C03662=1159.444,359.025,-79.936,-176.298,9.017,148.740
C03663=1159.448,358.778,-79.901,-176.300,9.013,148.740
C03664=1159.452,358.530,-79.866,-176.303,9.010,148.739
C03665=1159.456,358.283,-79.832,-176.305,9.006,148.739
C03666=1159.460,358.035,-79.798,-176.307,9.002,148.739
C03667=1159.465,357.787,-79.763,-176.310,8.998,148.739
C03668=1159.467,357.540,-79.728,-176.313,8.995,148.738
C03669=1159.472,357.292,-79.694,-176.315,8.990,148.738
C03670=1159.476,357.044,-79.659,-176.317,8.987,148.738
C03671=1159.480,356.797,-79.625,-176.320,8.983,148.737
C03672=1159.484,356.549,-79.590,-176.322,8.979,148.737
C03673=1159.488,356.302,-79.556,-176.325,8.975,148.737
C03674=1159.492,356.054,-79.521,-176.327,8.972,148.736
C03675=1159.496,355.806,-79.487,-176.330,8.968,148.736
C03676=1159.499,355.559,-79.453,-176.332,8.964,148.736
C03677=1159.504,355.311,-79.418,-176.335,8.960,148.736
C03678=1159.508,355.064,-79.384,-176.337,8.957,148.735
C03679=1159.512,354.816,-79.350,-176.340,8.953,148.735
C03680=1159.516,354.569,-79.315,-176.342,8.949,148.735
C03681=1159.520,354.321,-79.281,-176.344,8.946,148.734
C03682=1159.524,354.073,-79.246,-176.347,8.942,148.734
C03683=1159.527,353.826,-79.212,-176.349,8.938,148.734
C03684=1159.532,353.578,-79.178,-176.352,8.934,148.733
C03685=1159.536,353.331,-79.144,-176.354,8.931,148.733
C03686=1159.540,353.083,-79.109,-176.357,8.926,148.733
C03687=1159.544,352.836,-79.075,-176.359,8.923,148.733
C03688=1159.548,352.588,-79.040,-176.362,8.919,148.732
C03689=1159.552,352.340,-79.007,-176.364,8.915,148.732
C03690=1159.556,352.093,-78.973,-176.366,8.912,148.732
C03691=1159.559,351.845,-78.938,-176.369,8.908,148.732
C03692=1159.564,351.597,-78.904,-176.372,8.905,148.731
C03693=1159.568,351.350,-78.870,-176.374,8.900,148.731
C03694=1159.571,351.102,-78.837,-176.376,8.897,148.731
C03695=1159.576,350.854,-78.802,-176.379,8.894,148.731
C03696=1159.579,350.607,-78.768,-176.382,8.890,148.730
C03697=1159.584,350.359,-78.733,-176.384,8.886,148.730
C03698=1159.588,350.111,-78.700,-176.387,8.882,148.730
C03699=1159.592,349.863,-78.665,-176.389,8.879,148.729
C03700=1159.596,349.616,-78.632,-176.391,8.875,148.729
C03701=1159.600,349.368,-78.598,-176.394,8.871,148.729
C03702=1159.604,349.121,-78.564,-176.396,8.868,148.729
C03703=1159.608,348.873,-78.530,-176.399,8.864,148.728
C03704=1159.612,348.625,-78.496,-176.401,8.861,148.728
C03705=1159.616,348.378,-78.462,-176.404,8.856,148.728
C03706=1159.620,348.130,-78.428,-176.406,8.853,148.728
C03707=1159.624,347.883,-78.395,-176.408,8.850,148.727
C03708=1159.628,347.635,-78.360,-176.411,8.846,148.727
C03709=1159.632,347.387,-78.327,-176.414,8.842,148.727
C03710=1159.636,347.140,-78.293,-176.416,8.838,148.727
C03711=1159.641,346.892,-78.259,-176.419,8.835,148.726
C03712=1159.644,346.644,-78.225,-176.421,8.832,148.726
C03713=1159.649,346.397,-78.192,-176.423,8.827,148.726
C03714=1159.652,346.149,-78.158,-176.426,8.824,148.726
C03715=1159.657,345.901,-78.124,-176.428,8.821,148.725
C03716=1159.660,345.654,-78.090,-176.431,8.817,148.725
C03717=1159.665,345.406,-78.057,-176.433,8.813,148.725
C03718=1159.668,345.158,-78.023,-176.436,8.809,148.725
C03719=1159.673,344.910,-77.989,-176.438,8.806,148.724
C03720=1159.677,344.662,-77.956,-176.441,8.803,148.724
C03721=1159.681,344.415,-77.922,-176.444,8.798,148.724
C03722=1159.685,344.168,-77.889,-176.446,8.795,148.724
C03723=1159.689,343.919,-77.854,-176.448,8.792,148.724
C03724=1159.693,343.672,-77.821,-176.451,8.788,148.723
C03725=1159.697,343.424,-77.788,-176.453,8.785,148.723
C03726=1159.701,343.177,-77.754,-176.456,8.780,148.723
C03727=1159.705,342.929,-77.721,-176.458,8.777,148.722
C03728=1159.709,342.681,-77.687,-176.461,8.774,148.722
C03729=1159.713,342.433,-77.653,-176.463,8.769,148.722
C03730=1159.717,342.186,-77.619,-176.466,8.766,148.722
C03731=1159.721,341.938,-77.586,-176.468,8.763,148.722
C03732=1159.726,341.690,-77.553,-176.471,8.759,148.721
C03733=1159.730,341.442,-77.520,-176.473,8.755,148.721
C03734=1159.734,341.195,-77.486,-176.475,8.752,148.721
C03735=1159.738,340.948,-77.453,-176.478,8.748,148.721
C03736=1159.741,340.699,-77.419,-176.481,8.745,148.720
C03737=1159.745,340.451,-77.386,-176.483,8.741,148.720
C03738=1159.749,340.204,-77.353,-176.486,8.737,148.720
C03739=1159.755,339.924,-77.315,-176.489,8.733,148.720
C03740=1159.759,339.644,-77.278,-176.492,8.729,148.719
C03741=1159.764,339.365,-77.240,-176.494,8.726,148.719
C03742=1159.769,339.085,-77.202,-176.497,8.722,148.719
C03743=1159.772,338.837,-77.169,-176.500,8.718,148.719
C03744=1159.776,338.589,-77.136,-176.502,8.714,148.718
C03745=1159.780,338.341,-77.103,-176.504,8.711,148.718
C03746=1159.785,338.093,-77.069,-176.507,8.707,148.718
C03747=1159.789,337.846,-77.036,-176.509,8.704,148.718
C03748=1159.793,337.598,-77.003,-176.512,8.700,148.718
C03749=1159.797,337.350,-76.970,-176.515,8.696,148.717
C03750=1159.801,337.102,-76.937,-176.517,8.693,148.717
C03751=1159.805,336.855,-76.904,-176.519,8.690,148.717
C03752=1159.809,336.607,-76.871,-176.523,8.686,148.717
C03753=1159.813,336.360,-76.838,-176.525,8.683,148.717
C03754=1159.817,336.112,-76.805,-176.527,8.679,148.717
C03755=1159.821,335.864,-76.772,-176.530,8.675,148.716
C03756=1159.825,335.616,-76.739,-176.532,8.672,148.716
C03757=1159.829,335.369,-76.705,-176.535,8.669,148.716
C03758=1159.834,335.120,-76.673,-176.537,8.665,148.716
C03759=1159.838,334.873,-76.640,-176.540,8.661,148.715
C03760=1159.841,334.625,-76.607,-176.542,8.658,148.715
C03761=1159.845,334.377,-76.574,-176.544,8.655,148.715
C03762=1159.850,334.130,-76.541,-176.547,8.651,148.715
C03763=1159.854,333.881,-76.508,-176.550,8.647,148.715
C03764=1159.858,333.634,-76.475,-176.552,8.644,148.714
C03765=1159.862,333.386,-76.442,-176.555,8.640,148.714
C03766=1159.866,333.138,-76.410,-176.558,8.637,148.714
C03767=1159.870,332.890,-76.377,-176.560,8.634,148.714
C03768=1159.874,332.642,-76.344,-176.562,8.630,148.714
C03769=1159.878,332.395,-76.311,-176.565,8.626,148.713
C03770=1159.883,332.147,-76.278,-176.567,8.623,148.713
C03771=1159.886,331.899,-76.246,-176.570,8.620,148.713
C03772=1159.890,331.651,-76.213,-176.573,8.616,148.713
C03773=1159.895,331.403,-76.179,-176.575,8.612,148.713
C03774=1159.898,331.155,-76.148,-176.578,8.609,148.713
C03775=1159.902,330.908,-76.114,-176.580,8.606,148.712
C03776=1159.907,330.659,-76.082,-176.583,8.602,148.712
C03777=1159.911,330.412,-76.049,-176.585,8.599,148.712
C03778=1159.915,330.165,-76.017,-176.587,8.595,148.712
C03779=1159.919,329.917,-75.984,-176.590,8.592,148.712
C03780=1159.924,329.669,-75.951,-176.593,8.588,148.711
C03781=1159.927,329.421,-75.919,-176.595,8.585,148.711
C03782=1159.931,329.173,-75.886,-176.598,8.582,148.711
C03783=1159.936,328.925,-75.854,-176.601,8.578,148.711
C03784=1159.939,328.677,-75.821,-176.603,8.574,148.711
C03785=1159.944,328.429,-75.789,-176.605,8.571,148.711
C03786=1159.948,328.182,-75.756,-176.607,8.568,148.710
C03787=1159.952,327.934,-75.724,-176.611,8.564,148.710
C03788=1159.956,327.686,-75.691,-176.613,8.561,148.710
C03789=1159.960,327.438,-75.659,-176.615,8.557,148.710
C03790=1159.964,327.190,-75.627,-176.618,8.554,148.710
C03791=1159.969,326.942,-75.593,-176.621,8.550,148.709
C03792=1159.973,326.695,-75.562,-176.623,8.547,148.709
C03793=1159.977,326.447,-75.529,-176.626,8.544,148.709
C03794=1159.981,326.199,-75.497,-176.628,8.541,148.709
C03795=1159.985,325.951,-75.465,-176.631,8.536,148.709
C03796=1159.989,325.703,-75.432,-176.633,8.533,148.709
C03797=1159.993,325.455,-75.400,-176.636,8.530,148.709
C03798=1159.997,325.207,-75.368,-176.638,8.527,148.708
C03799=1160.002,324.959,-75.336,-176.641,8.523,148.708
C03800=1160.005,324.712,-75.303,-176.643,8.520,148.708
C03801=1160.010,324.463,-75.271,-176.646,8.517,148.708
C03802=1160.013,324.215,-75.239,-176.648,8.513,148.708
C03803=1160.018,323.968,-75.206,-176.651,8.510,148.708
C03804=1160.022,323.720,-75.174,-176.654,8.506,148.707
C03805=1160.026,323.472,-75.142,-176.656,8.503,148.707
C03806=1160.030,323.224,-75.110,-176.659,8.500,148.707
C03807=1160.035,322.976,-75.078,-176.661,8.496,148.707
C03808=1160.039,322.728,-75.046,-176.664,8.492,148.707
C03809=1160.042,322.481,-75.013,-176.666,8.489,148.707
C03810=1160.047,322.232,-74.981,-176.669,8.486,148.707
C03811=1160.051,321.985,-74.949,-176.671,8.483,148.706
C03812=1160.055,321.737,-74.917,-176.674,8.479,148.706
C03813=1160.059,321.489,-74.885,-176.677,8.476,148.706
C03814=1160.063,321.241,-74.853,-176.679,8.472,148.706
C03815=1160.068,320.993,-74.821,-176.681,8.469,148.706
C03816=1160.071,320.745,-74.789,-176.684,8.466,148.706
C03817=1160.075,320.497,-74.758,-176.687,8.462,148.706
C03818=1160.080,320.249,-74.725,-176.689,8.459,148.705
C03819=1160.084,320.001,-74.694,-176.692,8.455,148.705
C03820=1160.088,319.753,-74.662,-176.694,8.452,148.705
C03821=1160.093,319.506,-74.630,-176.697,8.449,148.705
C03822=1160.096,319.257,-74.598,-176.700,8.445,148.705
C03823=1160.100,319.009,-74.566,-176.702,8.442,148.705
C03824=1160.105,318.762,-74.534,-176.705,8.439,148.705
C03825=1160.109,318.514,-74.502,-176.707,8.436,148.704
C03826=1160.113,318.266,-74.470,-176.709,8.432,148.704
C03827=1160.117,318.018,-74.439,-176.713,8.428,148.704
C03828=1160.121,317.770,-74.406,-176.715,8.425,148.704
C03829=1160.125,317.522,-74.374,-176.717,8.422,148.704
C03830=1160.130,317.274,-74.344,-176.720,8.419,148.704
C03831=1160.133,317.026,-74.312,-176.722,8.416,148.704
C03832=1160.137,316.778,-74.280,-176.725,8.412,148.703
C03833=1160.142,316.530,-74.248,-176.728,8.409,148.703
C03834=1160.146,316.282,-74.216,-176.730,8.405,148.703
C03835=1160.150,316.035,-74.185,-176.732,8.402,148.703
C03836=1160.154,315.786,-74.153,-176.735,8.399,148.703
C03837=1160.158,315.538,-74.122,-176.738,8.395,148.703
C03838=1160.163,315.291,-74.090,-176.740,8.392,148.703
C03839=1160.167,315.043,-74.058,-176.743,8.389,148.703
C03840=1160.171,314.795,-74.027,-176.745,8.385,148.702
C03841=1160.175,314.547,-73.995,-176.748,8.382,148.702
C03842=1160.179,314.299,-73.964,-176.750,8.379,148.702
C03843=1160.184,314.021,-73.929,-176.753,8.375,148.702
C03844=1160.189,313.744,-73.894,-176.757,8.371,148.702
C03845=1160.193,313.467,-73.858,-176.759,8.368,148.702
C03846=1160.198,313.190,-73.823,-176.762,8.364,148.702
C03847=1160.202,312.941,-73.792,-176.765,8.361,148.702
C03848=1160.206,312.694,-73.760,-176.767,8.358,148.701
C03849=1160.210,312.446,-73.728,-176.770,8.354,148.701
C03850=1160.215,312.198,-73.697,-176.773,8.351,148.701
C03851=1160.218,311.950,-73.666,-176.775,8.347,148.701
C03852=1160.223,311.702,-73.635,-176.778,8.344,148.701
C03853=1160.227,311.454,-73.603,-176.780,8.341,148.701
C03854=1160.231,311.206,-73.572,-176.783,8.338,148.701
C03855=1160.235,310.958,-73.540,-176.786,8.334,148.701
C03856=1160.240,310.710,-73.510,-176.788,8.331,148.700
C03857=1160.243,310.462,-73.478,-176.791,8.328,148.700
C03858=1160.248,310.214,-73.447,-176.793,8.324,148.700
C03859=1160.252,309.966,-73.415,-176.796,8.321,148.700
C03860=1160.256,309.718,-73.384,-176.798,8.318,148.700
C03861=1160.260,309.469,-73.353,-176.800,8.315,148.700
C03862=1160.264,309.222,-73.322,-176.804,8.311,148.700
C03863=1160.268,308.973,-73.291,-176.806,8.308,148.700
C03864=1160.273,308.726,-73.259,-176.809,8.305,148.700
C03865=1160.277,308.477,-73.228,-176.811,8.302,148.700
C03866=1160.281,308.229,-73.197,-176.814,8.299,148.700
C03867=1160.286,307.982,-73.166,-176.816,8.295,148.699
C03868=1160.290,307.733,-73.135,-176.818,8.292,148.699
C03869=1160.294,307.485,-73.104,-176.822,8.288,148.699
C03870=1160.298,307.237,-73.072,-176.824,8.285,148.699
C03871=1160.302,306.990,-73.042,-176.827,8.282,148.699
C03872=1160.307,306.742,-73.011,-176.829,8.279,148.699
C03873=1160.311,306.493,-72.980,-176.832,8.276,148.699
C03874=1160.315,306.246,-72.949,-176.834,8.272,148.699
C03875=1160.319,305.997,-72.917,-176.837,8.269,148.699
C03876=1160.323,305.749,-72.887,-176.839,8.266,148.699
C03877=1160.328,305.501,-72.856,-176.842,8.262,148.698
C03878=1160.331,305.253,-72.825,-176.845,8.259,148.698
C03879=1160.336,305.005,-72.794,-176.847,8.256,148.698
C03880=1160.340,304.757,-72.763,-176.850,8.253,148.698
C03881=1160.344,304.509,-72.732,-176.853,8.250,148.698
C03882=1160.349,304.261,-72.701,-176.855,8.247,148.698
C03883=1160.353,304.013,-72.671,-176.858,8.244,148.698
C03884=1160.357,303.765,-72.640,-176.860,8.240,148.698
C03885=1160.361,303.517,-72.609,-176.863,8.237,148.698
C03886=1160.366,303.269,-72.578,-176.866,8.233,148.698
C03887=1160.369,303.020,-72.548,-176.868,8.230,148.698
C03888=1160.374,302.772,-72.517,-176.871,8.227,148.697
C03889=1160.378,302.525,-72.486,-176.873,8.224,148.698
C03890=1160.382,302.276,-72.454,-176.876,8.221,148.697
C03891=1160.386,302.029,-72.424,-176.878,8.218,148.697
C03892=1160.391,301.781,-72.394,-176.881,8.215,148.697
C03893=1160.395,301.533,-72.363,-176.883,8.212,148.697
C03894=1160.399,301.284,-72.333,-176.886,8.208,148.697
C03895=1160.404,301.036,-72.302,-176.889,8.205,148.697
C03896=1160.408,300.788,-72.271,-176.891,8.201,148.697
C03897=1160.411,300.540,-72.241,-176.894,8.198,148.697
C03898=1160.416,300.292,-72.210,-176.896,8.195,148.697
C03899=1160.421,300.044,-72.179,-176.899,8.192,148.697
C03900=1160.425,299.796,-72.149,-176.901,8.189,148.697
C03901=1160.429,299.547,-72.118,-176.904,8.186,148.697
C03902=1160.433,299.299,-72.087,-176.907,8.183,148.696
C03903=1160.437,299.052,-72.057,-176.909,8.180,148.696
C03904=1160.442,298.803,-72.027,-176.912,8.177,148.696
C03905=1160.445,298.555,-71.997,-176.914,8.173,148.696
C03906=1160.450,298.307,-71.966,-176.918,8.170,148.696
C03907=1160.454,298.059,-71.935,-176.920,8.166,148.696
C03908=1160.458,297.811,-71.905,-176.923,8.163,148.696
C03909=1160.463,297.563,-71.875,-176.925,8.160,148.696
C03910=1160.467,297.314,-71.844,-176.928,8.157,148.696
C03911=1160.471,297.066,-71.813,-176.931,8.154,148.696
C03912=1160.475,296.818,-71.784,-176.933,8.151,148.696
C03913=1160.480,296.570,-71.753,-176.936,8.148,148.696
C03914=1160.484,296.322,-71.723,-176.938,8.145,148.696
C03915=1160.488,296.074,-71.692,-176.941,8.142,148.696
C03916=1160.492,295.826,-71.663,-176.943,8.138,148.695
C03917=1160.497,295.578,-71.632,-176.946,8.135,148.696
C03918=1160.500,295.330,-71.602,-176.948,8.132,148.696
C03919=1160.505,295.081,-71.572,-176.951,8.128,148.695
C03920=1160.509,294.834,-71.541,-176.954,8.125,148.695
C03921=1160.513,294.585,-71.512,-176.956,8.122,148.695
C03922=1160.517,294.337,-71.481,-176.959,8.119,148.695
C03923=1160.521,294.089,-71.451,-176.962,8.116,148.695
C03924=1160.526,293.841,-71.421,-176.964,8.113,148.695
C03925=1160.530,293.593,-71.390,-176.967,8.110,148.695
C03926=1160.534,293.345,-71.361,-176.970,8.107,148.695
C03927=1160.539,293.097,-71.330,-176.972,8.104,148.695
C03928=1160.543,292.848,-71.301,-176.975,8.101,148.695
C03929=1160.547,292.600,-71.270,-176.977,8.097,148.695
C03930=1160.551,292.351,-71.240,-176.980,8.094,148.695
C03931=1160.555,292.104,-71.210,-176.983,8.091,148.695
C03932=1160.560,291.855,-71.180,-176.985,8.088,148.695
C03933=1160.564,291.607,-71.150,-176.988,8.085,148.695
C03934=1160.568,291.359,-71.120,-176.990,8.082,148.695
C03935=1160.573,291.111,-71.090,-176.993,8.079,148.695
C03936=1160.577,290.863,-71.060,-176.995,8.076,148.695
C03937=1160.581,290.615,-71.031,-176.998,8.073,148.695
C03938=1160.585,290.367,-71.001,-177.001,8.069,148.694
C03939=1160.590,290.119,-70.970,-177.004,8.066,148.695
C03940=1160.594,289.870,-70.941,-177.007,8.063,148.695
C03941=1160.598,289.622,-70.912,-177.009,8.060,148.694
C03942=1160.603,289.374,-70.881,-177.012,8.057,148.694
C03943=1160.607,289.126,-70.851,-177.014,8.054,148.694
C03944=1160.611,288.878,-70.822,-177.017,8.051,148.694
C03945=1160.615,288.630,-70.792,-177.019,8.048,148.694
C03946=1160.619,288.382,-70.762,-177.022,8.045,148.694
C03947=1160.624,288.106,-70.729,-177.025,8.041,148.694
C03948=1160.628,287.831,-70.696,-177.028,8.038,148.694
C03949=1160.633,287.555,-70.663,-177.031,8.035,148.694
C03950=1160.638,287.281,-70.630,-177.034,8.031,148.694
C03951=1160.642,287.032,-70.601,-177.036,8.028,148.694
C03952=1160.647,286.784,-70.571,-177.039,8.025,148.694
C03953=1160.651,286.536,-70.541,-177.042,8.022,148.694
C03954=1160.656,286.289,-70.511,-177.044,8.018,148.694
C03955=1160.660,286.040,-70.482,-177.047,8.015,148.694
C03956=1160.664,285.792,-70.452,-177.050,8.012,148.694
C03957=1160.668,285.544,-70.423,-177.052,8.009,148.694
C03958=1160.672,285.296,-70.393,-177.055,8.006,148.694
C03959=1160.677,285.047,-70.363,-177.057,8.003,148.694
C03960=1160.681,284.799,-70.334,-177.060,8.000,148.694
C03961=1160.686,284.550,-70.304,-177.062,7.997,148.694
C03962=1160.690,284.302,-70.275,-177.065,7.994,148.694
C03963=1160.694,284.054,-70.246,-177.068,7.991,148.694
C03964=1160.698,283.806,-70.216,-177.071,7.988,148.694
C03965=1160.702,283.557,-70.187,-177.073,7.985,148.694
C03966=1160.707,283.309,-70.157,-177.076,7.982,148.694
C03967=1160.711,283.061,-70.128,-177.079,7.979,148.694
C03968=1160.716,282.813,-70.099,-177.081,7.976,148.694
C03969=1160.720,282.565,-70.069,-177.084,7.973,148.694
C03970=1160.724,282.317,-70.040,-177.086,7.970,148.694
C03971=1160.728,282.068,-70.010,-177.089,7.967,148.694
C03972=1160.732,281.820,-69.981,-177.092,7.964,148.694
C03973=1160.736,281.572,-69.951,-177.094,7.961,148.694
C03974=1160.741,281.324,-69.922,-177.097,7.958,148.694
C03975=1160.746,281.076,-69.894,-177.100,7.955,148.694
C03976=1160.750,280.827,-69.864,-177.102,7.952,148.694
C03977=1160.754,280.579,-69.835,-177.105,7.948,148.694
C03978=1160.758,280.331,-69.805,-177.108,7.945,148.694
C03979=1160.762,280.082,-69.776,-177.110,7.942,148.694
C03980=1160.767,279.834,-69.746,-177.113,7.940,148.694
C03981=1160.771,279.585,-69.718,-177.115,7.936,148.694
C03982=1160.776,279.338,-69.688,-177.118,7.933,148.694
C03983=1160.780,279.089,-69.659,-177.121,7.930,148.694
C03984=1160.784,278.841,-69.630,-177.124,7.927,148.694
C03985=1160.788,278.593,-69.601,-177.126,7.924,148.694
C03986=1160.792,278.344,-69.572,-177.128,7.922,148.694
C03987=1160.797,278.097,-69.543,-177.131,7.919,148.694
C03988=1160.801,277.848,-69.514,-177.134,7.916,148.694
C03989=1160.806,277.600,-69.485,-177.136,7.913,148.694
C03990=1160.810,277.351,-69.455,-177.139,7.910,148.694
C03991=1160.814,277.103,-69.427,-177.141,7.907,148.694
C03992=1160.818,276.855,-69.398,-177.144,7.904,148.694
C03993=1160.823,276.607,-69.369,-177.147,7.901,148.694
C03994=1160.827,276.358,-69.340,-177.150,7.898,148.694
C03995=1160.831,276.110,-69.310,-177.152,7.895,148.694
C03996=1160.836,275.862,-69.283,-177.155,7.892,148.694
C03997=1160.840,275.614,-69.253,-177.158,7.889,148.694
C03998=1160.844,275.365,-69.224,-177.160,7.886,148.694
C03999=1160.848,275.116,-69.195,-177.163,7.883,148.694
C04000=1160.852,274.869,-69.166,-177.166,7.880,148.694
C04001=1160.857,274.620,-69.138,-177.169,7.877,148.694
C04002=1160.861,274.372,-69.108,-177.171,7.874,148.694
C04003=1160.866,274.124,-69.080,-177.174,7.871,148.694
C04004=1160.870,273.876,-69.051,-177.176,7.868,148.694
C04005=1160.874,273.627,-69.022,-177.179,7.865,148.694
C04006=1160.878,273.379,-68.993,-177.182,7.862,148.694
C04007=1160.883,273.131,-68.965,-177.185,7.859,148.694
C04008=1160.887,272.882,-68.936,-177.187,7.857,148.694
C04009=1160.891,272.634,-68.907,-177.189,7.853,148.694
C04010=1160.896,272.386,-68.879,-177.192,7.851,148.694
C04011=1160.900,272.138,-68.850,-177.195,7.848,148.694
C04012=1160.904,271.889,-68.821,-177.197,7.845,148.694
C04013=1160.909,271.641,-68.793,-177.200,7.842,148.694
C04014=1160.913,271.393,-68.764,-177.203,7.839,148.694
C04015=1160.917,271.144,-68.735,-177.206,7.836,148.694
C04016=1160.922,270.896,-68.707,-177.208,7.833,148.694
C04017=1160.926,270.648,-68.678,-177.211,7.830,148.694
C04018=1160.931,270.399,-68.649,-177.214,7.827,148.694
C04019=1160.935,270.151,-68.621,-177.216,7.824,148.694
C04020=1160.939,269.902,-68.592,-177.219,7.821,148.694
C04021=1160.943,269.655,-68.564,-177.222,7.818,148.694
C04022=1160.948,269.406,-68.535,-177.224,7.816,148.694
C04023=1160.952,269.157,-68.507,-177.227,7.813,148.694
C04024=1160.957,268.909,-68.479,-177.230,7.810,148.695
C04025=1160.960,268.660,-68.451,-177.232,7.807,148.695
C04026=1160.965,268.413,-68.421,-177.235,7.804,148.695
C04027=1160.970,268.164,-68.393,-177.237,7.800,148.694
C04028=1160.974,267.916,-68.365,-177.240,7.798,148.695
C04029=1160.978,267.667,-68.336,-177.243,7.795,148.695
C04030=1160.982,267.419,-68.308,-177.246,7.792,148.695
C04031=1160.987,267.170,-68.280,-177.248,7.789,148.695
C04032=1160.991,266.922,-68.252,-177.251,7.786,148.695
C04033=1160.996,266.674,-68.223,-177.253,7.784,148.695
C04034=1161.000,266.426,-68.194,-177.256,7.781,148.695
C04035=1161.004,266.178,-68.167,-177.259,7.778,148.695
C04036=1161.008,265.929,-68.138,-177.262,7.775,148.695
C04037=1161.013,265.681,-68.110,-177.264,7.772,148.695
C04038=1161.017,265.432,-68.081,-177.267,7.769,148.695
C04039=1161.022,265.184,-68.054,-177.270,7.766,148.695
C04040=1161.026,264.935,-68.025,-177.273,7.763,148.695
C04041=1161.030,264.688,-67.997,-177.275,7.760,148.695
C04042=1161.034,264.439,-67.969,-177.278,7.757,148.695
C04043=1161.039,264.191,-67.941,-177.280,7.755,148.695
C04044=1161.043,263.942,-67.912,-177.283,7.752,148.695
C04045=1161.048,263.693,-67.885,-177.285,7.749,148.695
C04046=1161.052,263.445,-67.857,-177.288,7.746,148.695
C04047=1161.057,263.197,-67.829,-177.291,7.743,148.695
C04048=1161.061,262.948,-67.800,-177.294,7.740,148.695
C04049=1161.065,262.700,-67.772,-177.296,7.737,148.696
C04050=1161.069,262.452,-67.744,-177.299,7.734,148.696
C04051=1161.074,262.178,-67.713,-177.302,7.731,148.696
C04052=1161.080,261.905,-67.683,-177.305,7.728,148.696
C04053=1161.084,261.632,-67.652,-177.308,7.725,148.696
C04054=1161.089,261.359,-67.621,-177.311,7.721,148.696
C04055=1161.093,261.110,-67.593,-177.313,7.719,148.696
C04056=1161.097,260.862,-67.565,-177.316,7.716,148.696
C04057=1161.102,260.613,-67.537,-177.319,7.713,148.696
C04058=1161.106,260.365,-67.509,-177.321,7.710,148.696
C04059=1161.111,260.117,-67.482,-177.324,7.707,148.696
C04060=1161.114,259.868,-67.454,-177.327,7.704,148.696
C04061=1161.119,259.621,-67.426,-177.330,7.701,148.696
C04062=1161.124,259.371,-67.398,-177.332,7.699,148.696
C04063=1161.128,259.123,-67.370,-177.335,7.696,148.696
C04064=1161.132,258.875,-67.342,-177.337,7.693,148.696
C04065=1161.136,258.626,-67.315,-177.341,7.691,148.697
C04066=1161.141,258.378,-67.287,-177.343,7.688,148.697
C04067=1161.146,258.130,-67.259,-177.346,7.685,148.697
C04068=1161.150,257.881,-67.231,-177.349,7.682,148.697
C04069=1161.154,257.633,-67.203,-177.351,7.680,148.697
C04070=1161.158,257.384,-67.176,-177.354,7.677,148.697
C04071=1161.163,257.136,-67.148,-177.357,7.674,148.697
C04072=1161.167,256.888,-67.120,-177.359,7.671,148.697
C04073=1161.172,256.638,-67.092,-177.362,7.668,148.697
C04074=1161.176,256.391,-67.065,-177.365,7.665,148.697
C04075=1161.181,256.142,-67.038,-177.367,7.663,148.697
C04076=1161.185,255.894,-67.009,-177.370,7.660,148.697
C04077=1161.189,255.645,-66.982,-177.373,7.657,148.697
C04078=1161.194,255.397,-66.955,-177.375,7.654,148.698
C04079=1161.198,255.149,-66.928,-177.378,7.651,148.698
C04080=1161.202,254.900,-66.899,-177.381,7.648,148.698
C04081=1161.207,254.652,-66.872,-177.383,7.646,148.698
C04082=1161.211,254.403,-66.845,-177.386,7.643,148.698
C04083=1161.215,254.154,-66.817,-177.389,7.640,148.698
C04084=1161.220,253.906,-66.790,-177.391,7.637,148.698
C04085=1161.224,253.658,-66.762,-177.394,7.634,148.698
C04086=1161.229,253.410,-66.735,-177.397,7.632,148.698
C04087=1161.233,253.160,-66.708,-177.400,7.629,148.698
C04088=1161.237,252.913,-66.680,-177.402,7.627,148.698
C04089=1161.242,252.664,-66.653,-177.405,7.624,148.699
C04090=1161.246,252.415,-66.626,-177.408,7.621,148.699
C04091=1161.250,252.167,-66.598,-177.411,7.618,148.699
C04092=1161.255,251.918,-66.571,-177.413,7.616,148.699
C04093=1161.259,251.670,-66.544,-177.416,7.613,148.699
C04094=1161.264,251.422,-66.516,-177.418,7.610,148.699
C04095=1161.268,251.173,-66.488,-177.421,7.607,148.699
C04096=1161.273,250.924,-66.461,-177.424,7.604,148.699
C04097=1161.277,250.676,-66.434,-177.427,7.602,148.699
C04098=1161.282,250.428,-66.407,-177.429,7.599,148.699
C04099=1161.286,250.179,-66.379,-177.432,7.596,148.699
C04100=1161.290,249.930,-66.352,-177.435,7.593,148.700
C04101=1161.294,249.682,-66.326,-177.438,7.590,148.700
C04102=1161.299,249.434,-66.299,-177.440,7.588,148.700
C04103=1161.303,249.186,-66.271,-177.443,7.585,148.700
C04104=1161.308,248.937,-66.244,-177.445,7.582,148.700
C04105=1161.312,248.688,-66.216,-177.449,7.580,148.700
C04106=1161.317,248.440,-66.189,-177.451,7.577,148.700
C04107=1161.321,248.191,-66.162,-177.454,7.574,148.700
C04108=1161.325,247.943,-66.136,-177.456,7.572,148.700
C04109=1161.330,247.694,-66.109,-177.459,7.569,148.700
C04110=1161.334,247.446,-66.082,-177.462,7.566,148.700
C04111=1161.338,247.197,-66.054,-177.464,7.564,148.701
C04112=1161.343,246.948,-66.027,-177.467,7.561,148.701
C04113=1161.347,246.700,-66.001,-177.470,7.558,148.701
C04114=1161.352,246.452,-65.974,-177.473,7.555,148.701
C04115=1161.356,246.203,-65.946,-177.476,7.552,148.701
C04116=1161.361,245.955,-65.919,-177.478,7.550,148.701
C04117=1161.366,245.706,-65.892,-177.481,7.547,148.701
C04118=1161.370,245.458,-65.866,-177.483,7.544,148.701
C04119=1161.374,245.209,-65.839,-177.487,7.541,148.702
C04120=1161.378,244.960,-65.811,-177.489,7.539,148.702
C04121=1161.382,244.712,-65.785,-177.491,7.536,148.702
C04122=1161.387,244.464,-65.758,-177.494,7.533,148.702
C04123=1161.392,244.215,-65.731,-177.497,7.530,148.702
C04124=1161.395,243.967,-65.704,-177.499,7.528,148.702
C04125=1161.400,243.718,-65.677,-177.502,7.526,148.702
C04126=1161.405,243.470,-65.650,-177.505,7.523,148.702
C04127=1161.409,243.221,-65.624,-177.508,7.520,148.702
C04128=1161.414,242.973,-65.597,-177.510,7.518,148.703
C04129=1161.418,242.724,-65.570,-177.513,7.515,148.703
C04130=1161.422,242.476,-65.544,-177.516,7.512,148.703
C04131=1161.427,242.227,-65.517,-177.519,7.509,148.703
C04132=1161.432,241.978,-65.490,-177.521,7.507,148.703
C04133=1161.436,241.730,-65.464,-177.524,7.504,148.703
C04134=1161.440,241.482,-65.437,-177.527,7.501,148.703
C04135=1161.444,241.233,-65.410,-177.530,7.499,148.704
C04136=1161.449,240.984,-65.384,-177.532,7.496,148.704
C04137=1161.454,240.736,-65.357,-177.535,7.494,148.704
C04138=1161.458,240.488,-65.331,-177.538,7.491,148.704
C04139=1161.463,240.239,-65.304,-177.540,7.488,148.704
C04140=1161.467,239.990,-65.278,-177.543,7.486,148.704
C04141=1161.471,239.742,-65.251,-177.546,7.483,148.704
C04142=1161.475,239.494,-65.224,-177.549,7.480,148.704
C04143=1161.480,239.245,-65.198,-177.551,7.478,148.704
C04144=1161.484,238.996,-65.171,-177.554,7.475,148.705
C04145=1161.489,238.747,-65.145,-177.557,7.472,148.705
C04146=1161.494,238.499,-65.118,-177.560,7.469,148.705
C04147=1161.498,238.251,-65.092,-177.562,7.467,148.705
C04148=1161.502,238.002,-65.066,-177.565,7.465,148.705
C04149=1161.507,237.753,-65.039,-177.568,7.462,148.705
C04150=1161.511,237.504,-65.013,-177.570,7.460,148.705
C04151=1161.516,237.256,-64.986,-177.573,7.457,148.706
C04152=1161.520,237.007,-64.960,-177.576,7.454,148.706
C04153=1161.524,236.759,-64.933,-177.578,7.452,148.706
C04154=1161.529,236.510,-64.907,-177.581,7.449,148.706
C04155=1161.534,236.238,-64.878,-177.584,7.446,148.706
C04156=1161.538,235.967,-64.849,-177.587,7.443,148.706
C04157=1161.544,235.695,-64.821,-177.590,7.440,148.706
C04158=1161.548,235.423,-64.792,-177.593,7.438,148.707
C04159=1161.553,235.174,-64.766,-177.596,7.435,148.707
C04160=1161.557,234.927,-64.739,-177.598,7.432,148.707
C04161=1161.562,234.678,-64.714,-177.601,7.430,148.707
C04162=1161.567,234.429,-64.687,-177.604,7.427,148.707
C04163=1161.571,234.181,-64.661,-177.607,7.424,148.707
C04164=1161.575,233.932,-64.635,-177.609,7.422,148.707
C04165=1161.580,233.683,-64.609,-177.612,7.420,148.708
C04166=1161.584,233.435,-64.582,-177.615,7.417,148.708
C04167=1161.588,233.187,-64.557,-177.618,7.414,148.708
C04168=1161.593,232.937,-64.531,-177.620,7.412,148.708
C04169=1161.597,232.689,-64.504,-177.623,7.409,148.708
C04170=1161.602,232.440,-64.478,-177.626,7.406,148.708
C04171=1161.607,232.191,-64.452,-177.628,7.404,148.709
C04172=1161.610,231.943,-64.426,-177.631,7.401,148.709
C04173=1161.615,231.695,-64.400,-177.634,7.398,148.709
C04174=1161.620,231.446,-64.374,-177.636,7.396,148.709
C04175=1161.624,231.197,-64.348,-177.639,7.394,148.709
C04176=1161.628,230.949,-64.322,-177.642,7.391,148.709
C04177=1161.633,230.700,-64.296,-177.644,7.389,148.710
C04178=1161.637,230.452,-64.270,-177.647,7.386,148.710
C04179=1161.642,230.203,-64.244,-177.650,7.384,148.710
C04180=1161.647,229.954,-64.218,-177.653,7.381,148.710
C04181=1161.651,229.705,-64.193,-177.655,7.378,148.710
C04182=1161.655,229.458,-64.167,-177.658,7.376,148.710
C04183=1161.660,229.209,-64.141,-177.661,7.373,148.711
C04184=1161.665,228.960,-64.114,-177.664,7.370,148.711
C04185=1161.669,228.711,-64.089,-177.666,7.368,148.711
C04186=1161.673,228.462,-64.063,-177.669,7.366,148.711
C04187=1161.678,228.214,-64.038,-177.672,7.363,148.711
C04188=1161.682,227.965,-64.012,-177.675,7.361,148.711
C04189=1161.686,227.717,-63.986,-177.677,7.358,148.711
C04190=1161.691,227.468,-63.961,-177.681,7.355,148.712
C04191=1161.696,227.219,-63.934,-177.683,7.353,148.712
C04192=1161.700,226.971,-63.909,-177.686,7.350,148.712
C04193=1161.705,226.722,-63.883,-177.688,7.348,148.712
C04194=1161.709,226.474,-63.857,-177.691,7.345,148.712
C04195=1161.714,226.225,-63.832,-177.694,7.343,148.712
C04196=1161.718,225.976,-63.806,-177.696,7.341,148.713
C04197=1161.723,225.728,-63.781,-177.699,7.338,148.713
C04198=1161.727,225.479,-63.755,-177.702,7.335,148.713
C04199=1161.731,225.230,-63.729,-177.705,7.333,148.713
C04200=1161.736,224.982,-63.704,-177.707,7.330,148.713
C04201=1161.740,224.733,-63.678,-177.710,7.328,148.714
C04202=1161.744,224.485,-63.652,-177.713,7.325,148.714
C04203=1161.749,224.237,-63.627,-177.716,7.322,148.714
C04204=1161.754,223.987,-63.602,-177.718,7.321,148.714
C04205=1161.758,223.738,-63.576,-177.721,7.318,148.714
C04206=1161.763,223.490,-63.551,-177.723,7.316,148.714
C04207=1161.767,223.241,-63.525,-177.726,7.313,148.715
C04208=1161.771,222.993,-63.499,-177.729,7.310,148.715
C04209=1161.776,222.744,-63.474,-177.732,7.308,148.715
C04210=1161.781,222.495,-63.449,-177.735,7.305,148.715
C04211=1161.785,222.247,-63.423,-177.737,7.303,148.715
C04212=1161.790,221.998,-63.398,-177.740,7.301,148.716
C04213=1161.794,221.749,-63.372,-177.743,7.298,148.716
C04214=1161.799,221.501,-63.347,-177.746,7.296,148.716
C04215=1161.803,221.252,-63.321,-177.748,7.293,148.716
C04216=1161.808,221.004,-63.296,-177.751,7.291,148.716
C04217=1161.813,220.754,-63.271,-177.754,7.288,148.717
C04218=1161.817,220.505,-63.245,-177.756,7.286,148.717
C04219=1161.822,220.257,-63.220,-177.759,7.284,148.717
C04220=1161.826,220.008,-63.195,-177.762,7.281,148.717
C04221=1161.830,219.760,-63.170,-177.764,7.279,148.717
C04222=1161.834,219.511,-63.144,-177.767,7.276,148.718
C04223=1161.839,219.262,-63.119,-177.770,7.274,148.718
C04224=1161.844,219.014,-63.094,-177.773,7.271,148.718
C04225=1161.848,218.765,-63.068,-177.775,7.269,148.718
C04226=1161.853,218.516,-63.043,-177.778,7.266,148.718
C04227=1161.857,218.268,-63.018,-177.781,7.264,148.718
C04228=1161.862,218.019,-62.994,-177.783,7.261,148.719
C04229=1161.866,217.770,-62.968,-177.787,7.259,148.719
C04230=1161.871,217.522,-62.943,-177.789,7.257,148.719
C04231=1161.875,217.273,-62.917,-177.792,7.254,148.719
C04232=1161.880,217.024,-62.893,-177.794,7.252,148.719
C04233=1161.884,216.776,-62.868,-177.797,7.249,148.720
C04234=1161.889,216.527,-62.843,-177.800,7.247,148.720
C04235=1161.893,216.278,-62.817,-177.803,7.245,148.720
C04236=1161.898,216.030,-62.793,-177.806,7.242,148.720
C04237=1161.902,215.781,-62.767,-177.808,7.240,148.720
C04238=1161.907,215.532,-62.743,-177.811,7.237,148.721
C04239=1161.911,215.283,-62.717,-177.813,7.235,148.721
C04240=1161.916,215.035,-62.693,-177.817,7.232,148.721
C04241=1161.920,214.785,-62.668,-177.819,7.230,148.721
C04242=1161.925,214.537,-62.642,-177.822,7.228,148.722
C04243=1161.929,214.288,-62.618,-177.824,7.226,148.722
C04244=1161.934,214.040,-62.593,-177.827,7.223,148.722
C04245=1161.938,213.791,-62.568,-177.830,7.221,148.722
C04246=1161.943,213.542,-62.543,-177.833,7.218,148.722
C04247=1161.947,213.294,-62.518,-177.835,7.216,148.723
C04248=1161.952,213.045,-62.493,-177.838,7.213,148.723
C04249=1161.956,212.796,-62.469,-177.841,7.211,148.723
C04250=1161.961,212.547,-62.444,-177.844,7.209,148.723
C04251=1161.966,212.299,-62.419,-177.846,7.207,148.723
C04252=1161.970,212.050,-62.394,-177.849,7.204,148.724
C04253=1161.975,211.801,-62.369,-177.851,7.202,148.724
C04254=1161.979,211.553,-62.345,-177.855,7.199,148.724
C04255=1161.983,211.304,-62.320,-177.857,7.197,148.724
C04256=1161.988,211.055,-62.295,-177.860,7.195,148.725
C04257=1161.993,210.807,-62.271,-177.862,7.193,148.725
C04258=1161.997,210.557,-62.246,-177.866,7.190,148.725
C04259=1162.002,210.287,-62.219,-177.868,7.187,148.725
C04260=1162.007,210.016,-62.192,-177.872,7.184,148.725
C04261=1162.012,209.746,-62.165,-177.874,7.182,148.726
C04262=1162.017,209.476,-62.139,-177.877,7.180,148.726
C04263=1162.021,209.227,-62.114,-177.880,7.177,148.726
C04264=1162.026,208.978,-62.090,-177.883,7.175,148.726
C04265=1162.031,208.730,-62.065,-177.886,7.172,148.727
C04266=1162.035,208.480,-62.040,-177.888,7.170,148.727
C04267=1162.040,208.232,-62.016,-177.891,7.168,148.727
C04268=1162.045,207.983,-61.992,-177.893,7.166,148.727
C04269=1162.048,207.734,-61.967,-177.897,7.163,148.728
C04270=1162.053,207.486,-61.942,-177.899,7.161,148.728
C04271=1162.058,207.237,-61.918,-177.902,7.159,148.728
C04272=1162.062,206.988,-61.893,-177.904,7.156,148.728
C04273=1162.067,206.739,-61.869,-177.907,7.154,148.728
C04274=1162.072,206.491,-61.844,-177.910,7.151,148.729
C04275=1162.076,206.242,-61.820,-177.912,7.150,148.729
C04276=1162.081,205.992,-61.796,-177.915,7.147,148.729
C04277=1162.085,205.744,-61.772,-177.918,7.145,148.729
C04278=1162.090,205.495,-61.747,-177.921,7.142,148.730
C04279=1162.094,205.246,-61.722,-177.923,7.140,148.730
C04280=1162.099,204.998,-61.698,-177.927,7.138,148.730
C04281=1162.104,204.749,-61.674,-177.929,7.136,148.730
C04282=1162.108,204.501,-61.650,-177.932,7.133,148.731
C04283=1162.112,204.251,-61.625,-177.934,7.131,148.731
C04284=1162.117,204.003,-61.600,-177.937,7.129,148.731
C04285=1162.122,203.754,-61.576,-177.940,7.126,148.731
C04286=1162.126,203.505,-61.553,-177.942,7.124,148.731
C04287=1162.131,203.256,-61.528,-177.946,7.122,148.732
C04288=1162.135,203.007,-61.504,-177.948,7.120,148.732
C04289=1162.140,202.759,-61.480,-177.951,7.117,148.732
C04290=1162.145,202.510,-61.455,-177.953,7.115,148.732
C04291=1162.149,202.261,-61.432,-177.957,7.112,148.733
C04292=1162.153,202.012,-61.407,-177.959,7.110,148.733
C04293=1162.158,201.764,-61.383,-177.961,7.109,148.733
C04294=1162.163,201.515,-61.359,-177.965,7.106,148.734
C04295=1162.167,201.266,-61.335,-177.967,7.104,148.734
C04296=1162.172,201.018,-61.311,-177.970,7.101,148.734
C04297=1162.176,200.768,-61.287,-177.972,7.099,148.734
C04298=1162.181,200.520,-61.262,-177.976,7.097,148.734
C04299=1162.185,200.271,-61.239,-177.978,7.095,148.735
C04300=1162.190,200.022,-61.215,-177.981,7.093,148.735
C04301=1162.194,199.774,-61.191,-177.984,7.090,148.735
C04302=1162.200,199.524,-61.167,-177.986,7.088,148.735
C04303=1162.203,199.275,-61.142,-177.989,7.085,148.736
C04304=1162.208,199.026,-61.119,-177.992,7.084,148.736
C04305=1162.213,198.778,-61.095,-177.995,7.081,148.736
C04306=1162.217,198.530,-61.071,-177.997,7.079,148.736
C04307=1162.222,198.280,-61.047,-178.000,7.077,148.737
C04308=1162.227,198.032,-61.023,-178.003,7.074,148.737
C04309=1162.231,197.783,-60.999,-178.005,7.072,148.737
C04310=1162.236,197.534,-60.975,-178.008,7.070,148.737
C04311=1162.240,197.285,-60.952,-178.011,7.068,148.738
C04312=1162.244,197.036,-60.927,-178.013,7.066,148.738
C04313=1162.249,196.788,-60.903,-178.016,7.063,148.738
C04314=1162.253,196.539,-60.880,-178.019,7.061,148.739
C04315=1162.259,196.289,-60.856,-178.022,7.058,148.739
C04316=1162.263,196.041,-60.832,-178.025,7.057,148.739
C04317=1162.268,195.792,-60.809,-178.027,7.055,148.739
C04318=1162.272,195.544,-60.785,-178.030,7.052,148.739
C04319=1162.277,195.294,-60.761,-178.033,7.050,148.740
C04320=1162.281,195.046,-60.737,-178.035,7.048,148.740
C04321=1162.286,194.797,-60.714,-178.038,7.045,148.740
C04322=1162.291,194.549,-60.690,-178.041,7.044,148.741
C04323=1162.295,194.300,-60.666,-178.044,7.041,148.741
C04324=1162.299,194.050,-60.643,-178.046,7.039,148.741
C04325=1162.304,193.801,-60.619,-178.049,7.037,148.741
C04326=1162.308,193.552,-60.595,-178.052,7.034,148.742
C04327=1162.313,193.303,-60.572,-178.054,7.033,148.742
C04328=1162.318,193.055,-60.548,-178.058,7.030,148.742
C04329=1162.322,192.806,-60.524,-178.060,7.028,148.742
C04330=1162.327,192.557,-60.501,-178.063,7.026,148.743
C04331=1162.331,192.309,-60.477,-178.066,7.024,148.743
C04332=1162.336,192.059,-60.454,-178.068,7.021,148.743
C04333=1162.341,191.810,-60.430,-178.071,7.020,148.744
C04334=1162.345,191.561,-60.407,-178.074,7.017,148.744
C04335=1162.350,191.313,-60.383,-178.076,7.015,148.744
C04336=1162.355,191.064,-60.359,-178.079,7.013,148.744
C04337=1162.359,190.815,-60.336,-178.082,7.011,148.745
C04338=1162.365,190.567,-60.313,-178.084,7.009,148.745
C04339=1162.369,190.318,-60.289,-178.087,7.007,148.745
C04340=1162.374,190.069,-60.266,-178.090,7.004,148.745
C04341=1162.378,189.820,-60.242,-178.092,7.002,148.746
C04342=1162.382,189.571,-60.220,-178.096,7.000,148.746
C04343=1162.387,189.322,-60.196,-178.098,6.998,148.746
C04344=1162.392,189.073,-60.173,-178.101,6.996,148.746
C04345=1162.396,188.824,-60.149,-178.104,6.993,148.747
C04346=1162.401,188.576,-60.125,-178.107,6.991,148.747
C04347=1162.406,188.327,-60.102,-178.109,6.989,148.747
C04348=1162.410,188.078,-60.079,-178.112,6.987,148.748
C04349=1162.414,187.829,-60.056,-178.115,6.985,148.748
C04350=1162.419,187.580,-60.033,-178.117,6.983,148.748
C04351=1162.424,187.331,-60.009,-178.120,6.980,148.748
C04352=1162.429,187.083,-59.986,-178.123,6.978,148.749
C04353=1162.434,186.834,-59.963,-178.126,6.977,148.749
C04354=1162.438,186.585,-59.939,-178.128,6.974,148.749
C04355=1162.442,186.336,-59.917,-178.131,6.972,148.750
C04356=1162.447,186.087,-59.893,-178.134,6.970,148.750
C04357=1162.452,185.838,-59.870,-178.136,6.968,148.750
C04358=1162.456,185.589,-59.847,-178.139,6.966,148.750
C04359=1162.460,185.340,-59.824,-178.142,6.964,148.751
C04360=1162.465,185.091,-59.800,-178.145,6.962,148.751
C04361=1162.470,184.843,-59.777,-178.147,6.959,148.751
C04362=1162.475,184.594,-59.754,-178.150,6.957,148.752
C04363=1162.480,184.324,-59.730,-178.153,6.955,148.752
C04364=1162.485,184.054,-59.705,-178.156,6.953,148.752
C04365=1162.490,183.785,-59.680,-178.159,6.950,148.753
C04366=1162.495,183.515,-59.655,-178.162,6.949,148.753
C04367=1162.499,183.266,-59.632,-178.165,6.946,148.753
C04368=1162.504,183.017,-59.608,-178.167,6.944,148.754
C04369=1162.508,182.768,-59.586,-178.170,6.942,148.754
C04370=1162.513,182.519,-59.562,-178.173,6.939,148.754
C04371=1162.518,182.270,-59.539,-178.176,6.938,148.754
C04372=1162.522,182.022,-59.517,-178.178,6.936,148.755
C04373=1162.527,181.773,-59.494,-178.181,6.934,148.755
C04374=1162.532,181.524,-59.471,-178.184,6.931,148.755
C04375=1162.536,181.275,-59.448,-178.186,6.929,148.756
C04376=1162.541,181.027,-59.425,-178.189,6.928,148.756
C04377=1162.545,180.777,-59.403,-178.192,6.925,148.756
C04378=1162.550,180.528,-59.379,-178.195,6.923,148.756
C04379=1162.555,180.279,-59.356,-178.197,6.921,148.757
C04380=1162.559,180.030,-59.334,-178.200,6.919,148.757
C04381=1162.564,179.782,-59.311,-178.203,6.917,148.757
C04382=1162.568,179.533,-59.288,-178.206,6.915,148.758
C04383=1162.573,179.284,-59.265,-178.208,6.913,148.758
C04384=1162.577,179.034,-59.243,-178.211,6.911,148.758
C04385=1162.583,178.786,-59.220,-178.214,6.909,148.759
C04386=1162.587,178.537,-59.198,-178.217,6.907,148.759
C04387=1162.592,178.288,-59.174,-178.219,6.905,148.759
C04388=1162.596,178.040,-59.152,-178.222,6.903,148.760
C04389=1162.601,177.790,-59.129,-178.225,6.900,148.760
C04390=1162.605,177.541,-59.107,-178.228,6.899,148.760
C04391=1162.610,177.292,-59.084,-178.230,6.897,148.761
C04392=1162.615,177.044,-59.062,-178.233,6.894,148.761
C04393=1162.619,176.795,-59.038,-178.236,6.892,148.761
C04394=1162.624,176.545,-59.016,-178.238,6.891,148.761
C04395=1162.629,176.297,-58.993,-178.241,6.889,148.762
C04396=1162.633,176.048,-58.971,-178.243,6.887,148.762
C04397=1162.638,175.799,-58.948,-178.247,6.884,148.762
C04398=1162.643,175.550,-58.926,-178.249,6.882,148.763
C04399=1162.647,175.301,-58.903,-178.252,6.881,148.763
C04400=1162.652,175.052,-58.881,-178.255,6.879,148.763
C04401=1162.657,174.803,-58.858,-178.257,6.876,148.764
C04402=1162.661,174.554,-58.836,-178.260,6.874,148.764
C04403=1162.665,174.305,-58.813,-178.263,6.872,148.764
C04404=1162.671,174.056,-58.791,-178.266,6.871,148.765
C04405=1162.675,173.807,-58.769,-178.269,6.868,148.765
C04406=1162.680,173.558,-58.745,-178.271,6.866,148.765
C04407=1162.685,173.309,-58.724,-178.274,6.864,148.765
C04408=1162.689,173.061,-58.701,-178.276,6.862,148.766
C04409=1162.694,172.812,-58.678,-178.280,6.860,148.766
C04410=1162.699,172.562,-58.656,-178.282,6.858,148.767
C04411=1162.702,172.314,-58.634,-178.285,6.856,148.767
C04412=1162.708,172.065,-58.611,-178.287,6.854,148.767
C04413=1162.712,171.815,-58.589,-178.290,6.853,148.767
C04414=1162.717,171.567,-58.567,-178.293,6.850,148.768
C04415=1162.722,171.318,-58.544,-178.296,6.848,148.768
C04416=1162.726,171.068,-58.522,-178.299,6.846,148.769
C04417=1162.731,170.820,-58.501,-178.301,6.845,148.769
C04418=1162.736,170.571,-58.477,-178.303,6.843,148.769
C04419=1162.741,170.322,-58.456,-178.307,6.840,148.769
C04420=1162.745,170.073,-58.433,-178.309,6.838,148.770
C04421=1162.750,169.824,-58.412,-178.312,6.837,148.770
C04422=1162.754,169.575,-58.388,-178.315,6.835,148.770
C04423=1162.759,169.326,-58.367,-178.318,6.833,148.771
C04424=1162.764,169.077,-58.345,-178.320,6.830,148.771
C04425=1162.768,168.828,-58.323,-178.323,6.828,148.771
C04426=1162.773,168.579,-58.300,-178.326,6.827,148.772
C04427=1162.777,168.330,-58.278,-178.328,6.825,148.772
C04428=1162.782,168.081,-58.256,-178.331,6.823,148.772
C04429=1162.787,167.832,-58.234,-178.334,6.821,148.773
C04430=1162.791,167.583,-58.212,-178.337,6.819,148.773
C04431=1162.796,167.334,-58.190,-178.339,6.817,148.773
C04432=1162.801,167.085,-58.168,-178.342,6.815,148.774
C04433=1162.806,166.836,-58.146,-178.345,6.813,148.774
C04434=1162.810,166.587,-58.124,-178.347,6.811,148.774
C04435=1162.815,166.338,-58.102,-178.351,6.809,148.775
C04436=1162.820,166.089,-58.080,-178.353,6.807,148.775
C04437=1162.824,165.840,-58.057,-178.356,6.805,148.776
C04438=1162.829,165.591,-58.035,-178.359,6.804,148.776
C04439=1162.833,165.342,-58.013,-178.361,6.802,148.776
C04440=1162.838,165.093,-57.992,-178.364,6.800,148.776
C04441=1162.843,164.845,-57.970,-178.367,6.797,148.777
C04442=1162.847,164.595,-57.948,-178.370,6.796,148.777
C04443=1162.852,164.347,-57.926,-178.372,6.794,148.778
C04444=1162.857,164.097,-57.904,-178.375,6.792,148.778
C04445=1162.862,163.848,-57.883,-178.378,6.790,148.778
C04446=1162.866,163.599,-57.861,-178.380,6.789,148.779
C04447=1162.871,163.350,-57.839,-178.383,6.786,148.779
C04448=1162.876,163.101,-57.817,-178.386,6.784,148.779
C04449=1162.881,162.852,-57.795,-178.389,6.782,148.780
C04450=1162.886,162.603,-57.773,-178.391,6.780,148.780
C04451=1162.890,162.354,-57.751,-178.394,6.779,148.780
C04452=1162.895,162.105,-57.730,-178.397,6.777,148.781
C04453=1162.899,161.856,-57.708,-178.399,6.775,148.781
C04454=1162.904,161.607,-57.686,-178.403,6.773,148.781
C04455=1162.909,161.358,-57.665,-178.405,6.771,148.782
C04456=1162.913,161.109,-57.643,-178.408,6.769,148.782
C04457=1162.918,160.860,-57.621,-178.410,6.767,148.782
C04458=1162.922,160.611,-57.599,-178.413,6.765,148.783
C04459=1162.927,160.362,-57.578,-178.416,6.763,148.783
C04460=1162.933,160.113,-57.557,-178.418,6.762,148.783
C04461=1162.937,159.863,-57.535,-178.422,6.759,148.784
C04462=1162.941,159.615,-57.513,-178.424,6.757,148.784
C04463=1162.946,159.366,-57.492,-178.427,6.756,148.784
C04464=1162.950,159.117,-57.470,-178.430,6.754,148.785
C04465=1162.955,158.868,-57.449,-178.432,6.752,148.785
C04466=1162.960,158.619,-57.427,-178.435,6.750,148.786
C04467=1162.966,158.350,-57.404,-178.438,6.749,148.786
C04468=1162.970,158.081,-57.380,-178.441,6.746,148.786
C04469=1162.976,157.812,-57.357,-178.444,6.744,148.787
C04470=1162.980,157.543,-57.334,-178.447,6.742,148.787
C04471=1162.985,157.294,-57.312,-178.450,6.740,148.787
C04472=1162.990,157.044,-57.291,-178.452,6.738,148.788
C04473=1162.995,156.796,-57.269,-178.455,6.737,148.788
C04474=1162.999,156.547,-57.248,-178.458,6.735,148.789
C04475=1163.003,156.298,-57.227,-178.460,6.733,148.789
C04476=1163.008,156.049,-57.205,-178.463,6.731,148.789
C04477=1163.013,155.800,-57.184,-178.466,6.730,148.790
C04478=1163.018,155.551,-57.163,-178.469,6.728,148.790
C04479=1163.022,155.302,-57.141,-178.471,6.726,148.790
C04480=1163.028,155.052,-57.120,-178.474,6.724,148.791
C04481=1163.032,154.804,-57.099,-178.477,6.722,148.791
C04482=1163.037,154.555,-57.078,-178.479,6.720,148.791
C04483=1163.041,154.305,-57.056,-178.482,6.718,148.792
C04484=1163.046,154.056,-57.035,-178.485,6.716,148.792
C04485=1163.051,153.808,-57.013,-178.487,6.715,148.792
C04486=1163.056,153.559,-56.993,-178.490,6.713,148.793
C04487=1163.060,153.309,-56.971,-178.493,6.711,148.793
C04488=1163.065,153.060,-56.950,-178.496,6.709,148.794
C04489=1163.070,152.811,-56.928,-178.498,6.708,148.794
C04490=1163.074,152.562,-56.908,-178.501,6.706,148.794
C04491=1163.080,152.313,-56.887,-178.504,6.704,148.795
C04492=1163.084,152.064,-56.864,-178.507,6.702,148.795
C04493=1163.088,151.815,-56.844,-178.510,6.700,148.796
C04494=1163.093,151.566,-56.822,-178.512,6.698,148.796
C04495=1163.098,151.317,-56.801,-178.515,6.696,148.796
C04496=1163.104,151.068,-56.780,-178.518,6.695,148.797
C04497=1163.107,150.819,-56.759,-178.520,6.693,148.797
C04498=1163.112,150.569,-56.738,-178.523,6.691,148.797
C04499=1163.117,150.320,-56.717,-178.526,6.689,148.798
C04500=1163.122,150.072,-56.696,-178.529,6.688,148.798
C04501=1163.127,149.823,-56.675,-178.531,6.686,148.799
C04502=1163.132,149.573,-56.654,-178.534,6.684,148.799
C04503=1163.135,149.324,-56.633,-178.537,6.682,148.799
C04504=1163.141,149.075,-56.612,-178.539,6.681,148.800
C04505=1163.145,148.826,-56.591,-178.542,6.679,148.800
C04506=1163.150,148.577,-56.570,-178.545,6.677,148.800
C04507=1163.155,148.328,-56.549,-178.547,6.675,148.801
C04508=1163.160,148.079,-56.528,-178.550,6.674,148.801
C04509=1163.165,147.830,-56.507,-178.553,6.672,148.802
C04510=1163.169,147.581,-56.487,-178.556,6.670,148.802
C04511=1163.173,147.332,-56.465,-178.559,6.668,148.802
C04512=1163.179,147.082,-56.444,-178.562,6.666,148.803
C04513=1163.183,146.833,-56.424,-178.564,6.664,148.803
C04514=1163.188,146.584,-56.403,-178.567,6.663,148.804
C04515=1163.193,146.335,-56.382,-178.570,6.661,148.804
C04516=1163.198,146.086,-56.361,-178.572,6.659,148.804
C04517=1163.202,145.838,-56.340,-178.575,6.657,148.805
C04518=1163.207,145.588,-56.319,-178.578,6.656,148.805
C04519=1163.212,145.339,-56.299,-178.580,6.654,148.805
C04520=1163.217,145.090,-56.278,-178.583,6.652,148.806
C04521=1163.221,144.841,-56.257,-178.586,6.650,148.806
C04522=1163.226,144.591,-56.236,-178.589,6.649,148.807
C04523=1163.230,144.342,-56.216,-178.591,6.647,148.807
C04524=1163.235,144.093,-56.195,-178.594,6.645,148.807
C04525=1163.240,143.844,-56.174,-178.597,6.643,148.808
C04526=1163.245,143.595,-56.153,-178.599,6.642,148.808
C04527=1163.249,143.346,-56.133,-178.602,6.640,148.809
C04528=1163.254,143.097,-56.113,-178.605,6.638,148.809
C04529=1163.259,142.848,-56.092,-178.607,6.636,148.809
C04530=1163.263,142.599,-56.071,-178.610,6.635,148.810
C04531=1163.269,142.349,-56.050,-178.613,6.633,148.810
C04532=1163.273,142.101,-56.030,-178.616,6.631,148.810
C04533=1163.278,141.851,-56.009,-178.618,6.630,148.811
C04534=1163.283,141.602,-55.989,-178.621,6.628,148.811
C04535=1163.287,141.353,-55.968,-178.624,6.626,148.812
C04536=1163.292,141.104,-55.947,-178.627,6.625,148.812
C04537=1163.297,140.855,-55.927,-178.630,6.623,148.813
C04538=1163.301,140.606,-55.907,-178.632,6.621,148.813
C04539=1163.306,140.357,-55.886,-178.635,6.620,148.813
C04540=1163.311,140.108,-55.865,-178.638,6.618,148.814
C04541=1163.315,139.859,-55.845,-178.640,6.616,148.814
C04542=1163.321,139.609,-55.825,-178.643,6.614,148.815
C04543=1163.325,139.360,-55.804,-178.646,6.613,148.815
C04544=1163.330,139.111,-55.784,-178.648,6.611,148.815
C04545=1163.335,138.862,-55.763,-178.651,6.609,148.816
C04546=1163.339,138.613,-55.743,-178.654,6.607,148.816
C04547=1163.344,138.364,-55.722,-178.657,6.606,148.816
C04548=1163.349,138.114,-55.702,-178.659,6.604,148.817
C04549=1163.354,137.866,-55.682,-178.662,6.602,148.817
C04550=1163.359,137.617,-55.662,-178.664,6.601,148.818
C04551=1163.364,137.368,-55.641,-178.667,6.600,148.818
C04552=1163.368,137.118,-55.621,-178.670,6.598,148.819
C04553=1163.373,136.869,-55.601,-178.673,6.596,148.819
C04554=1163.377,136.620,-55.580,-178.675,6.595,148.819
C04555=1163.383,136.371,-55.559,-178.678,6.593,148.820
C04556=1163.387,136.122,-55.540,-178.681,6.591,148.820
C04557=1163.392,135.873,-55.519,-178.684,6.590,148.821
C04558=1163.396,135.624,-55.499,-178.686,6.588,148.821
C04559=1163.401,135.374,-55.479,-178.689,6.586,148.821
C04560=1163.407,135.125,-55.459,-178.692,6.584,148.822
C04561=1163.411,134.877,-55.438,-178.694,6.583,148.822
C04562=1163.416,134.627,-55.419,-178.697,6.581,148.823
C04563=1163.420,134.378,-55.398,-178.700,6.580,148.823
C04564=1163.425,134.129,-55.378,-178.703,6.578,148.824
C04565=1163.430,133.879,-55.358,-178.706,6.576,148.824
C04566=1163.435,133.630,-55.337,-178.708,6.574,148.824
C04567=1163.440,133.381,-55.318,-178.711,6.573,148.825
C04568=1163.444,133.132,-55.298,-178.714,6.571,148.825
C04569=1163.449,132.883,-55.278,-178.716,6.570,148.826
C04570=1163.454,132.634,-55.258,-178.719,6.568,148.826
C04571=1163.459,132.365,-55.236,-178.722,6.566,148.827
C04572=1163.464,132.097,-55.214,-178.725,6.564,148.827
C04573=1163.470,131.828,-55.192,-178.728,6.563,148.827
C04574=1163.474,131.559,-55.171,-178.731,6.561,148.828
C04575=1163.479,131.310,-55.151,-178.733,6.559,148.828
C04576=1163.484,131.061,-55.132,-178.736,6.558,148.829
C04577=1163.489,130.813,-55.111,-178.739,6.556,148.829
C04578=1163.493,130.563,-55.092,-178.742,6.554,148.829
C04579=1163.499,130.314,-55.071,-178.745,6.553,148.830
C04580=1163.503,130.064,-55.051,-178.747,6.551,148.830
C04581=1163.508,129.816,-55.031,-178.749,6.550,148.831
C04582=1163.513,129.566,-55.011,-178.752,6.548,148.831
C04583=1163.518,129.317,-54.992,-178.755,6.547,148.831
C04584=1163.522,129.068,-54.971,-178.758,6.545,148.832
C04585=1163.528,128.819,-54.952,-178.761,6.543,148.832
C04586=1163.532,128.570,-54.932,-178.763,6.542,148.833
C04587=1163.537,128.320,-54.912,-178.766,6.540,148.833
C04588=1163.542,128.071,-54.892,-178.769,6.538,148.834
C04589=1163.547,127.823,-54.872,-178.772,6.537,148.834
C04590=1163.551,127.573,-54.853,-178.774,6.535,148.834
C04591=1163.556,127.323,-54.833,-178.776,6.534,148.835
C04592=1163.560,127.075,-54.813,-178.780,6.533,148.835
C04593=1163.566,126.826,-54.793,-178.782,6.531,148.836
C04594=1163.571,126.576,-54.774,-178.785,6.529,148.836
C04595=1163.574,126.327,-54.754,-178.788,6.527,148.837
C04596=1163.579,126.078,-54.734,-178.790,6.526,148.837
C04597=1163.584,125.829,-54.715,-178.793,6.524,148.837
C04598=1163.589,125.579,-54.695,-178.796,6.522,148.838
C04599=1163.594,125.331,-54.675,-178.798,6.522,148.839
C04600=1163.599,125.082,-54.656,-178.801,6.520,148.839
C04601=1163.604,124.832,-54.636,-178.804,6.518,148.839
C04602=1163.608,124.582,-54.616,-178.807,6.516,148.840
C04603=1163.614,124.334,-54.597,-178.809,6.515,148.840
C04604=1163.618,124.085,-54.577,-178.812,6.513,148.840
C04605=1163.622,123.835,-54.558,-178.815,6.512,148.841
C04606=1163.627,123.587,-54.538,-178.818,6.510,148.842
C04607=1163.632,123.337,-54.519,-178.820,6.509,148.842
C04608=1163.637,123.087,-54.499,-178.823,6.507,148.842
C04609=1163.642,122.839,-54.480,-178.825,6.506,148.843
C04610=1163.647,122.589,-54.460,-178.828,6.504,148.843
C04611=1163.652,122.340,-54.440,-178.831,6.503,148.844
C04612=1163.656,122.091,-54.421,-178.834,6.501,148.844
C04613=1163.661,121.842,-54.401,-178.837,6.499,148.845
C04614=1163.666,121.592,-54.382,-178.839,6.498,148.845
C04615=1163.671,121.343,-54.362,-178.842,6.496,148.845
C04616=1163.676,121.094,-54.343,-178.844,6.495,148.846
C04617=1163.680,120.845,-54.324,-178.848,6.493,148.846
C04618=1163.685,120.596,-54.304,-178.850,6.492,148.847
C04619=1163.690,120.346,-54.285,-178.853,6.490,148.847
C04620=1163.695,120.097,-54.265,-178.855,6.489,148.848
C04621=1163.699,119.848,-54.246,-178.858,6.487,148.848
C04622=1163.704,119.599,-54.227,-178.861,6.486,148.848
C04623=1163.709,119.350,-54.207,-178.864,6.484,148.849
C04624=1163.715,119.101,-54.188,-178.866,6.482,148.849
C04625=1163.719,118.852,-54.169,-178.869,6.481,148.850
C04626=1163.723,118.602,-54.149,-178.871,6.480,148.850
C04627=1163.729,118.353,-54.130,-178.874,6.478,148.851
C04628=1163.733,118.104,-54.111,-178.877,6.477,148.851
C04629=1163.738,117.855,-54.092,-178.880,6.475,148.852
C04630=1163.743,117.605,-54.072,-178.883,6.473,148.852
C04631=1163.748,117.357,-54.053,-178.885,6.472,148.852
C04632=1163.752,117.107,-54.034,-178.887,6.471,148.853
C04633=1163.758,116.858,-54.015,-178.891,6.469,148.853
C04634=1163.762,116.608,-53.995,-178.893,6.468,148.854
C04635=1163.767,116.360,-53.977,-178.896,6.466,148.854
C04636=1163.772,116.110,-53.957,-178.899,6.464,148.855
C04637=1163.776,115.861,-53.938,-178.901,6.463,148.855
C04638=1163.781,115.612,-53.919,-178.904,6.462,148.856
C04639=1163.786,115.362,-53.900,-178.907,6.460,148.856
C04640=1163.791,115.113,-53.881,-178.910,6.459,148.857
C04641=1163.796,114.864,-53.861,-178.912,6.457,148.857
C04642=1163.801,114.615,-53.842,-178.914,6.456,148.857
C04643=1163.805,114.365,-53.824,-178.918,6.455,148.858
C04644=1163.811,114.116,-53.805,-178.920,6.453,148.858
C04645=1163.815,113.868,-53.786,-178.923,6.451,148.859
C04646=1163.820,113.618,-53.766,-178.926,6.449,148.859
C04647=1163.826,113.368,-53.748,-178.928,6.449,148.860
C04648=1163.830,113.119,-53.729,-178.931,6.447,148.860
C04649=1163.835,112.870,-53.709,-178.934,6.445,148.861
C04650=1163.839,112.621,-53.690,-178.936,6.444,148.861
C04651=1163.845,112.372,-53.672,-178.939,6.442,148.861
C04652=1163.849,112.122,-53.653,-178.942,6.441,148.862
C04653=1163.854,111.873,-53.633,-178.945,6.440,148.862
C04654=1163.858,111.624,-53.615,-178.947,6.438,148.863
C04655=1163.864,111.375,-53.596,-178.950,6.436,148.863
C04656=1163.868,111.126,-53.578,-178.953,6.435,148.864
C04657=1163.873,110.876,-53.558,-178.955,6.434,148.864
C04658=1163.878,110.627,-53.539,-178.958,6.432,148.865
C04659=1163.883,110.377,-53.520,-178.961,6.431,148.865
C04660=1163.887,110.129,-53.502,-178.964,6.429,148.866
C04661=1163.893,109.879,-53.483,-178.966,6.428,148.866
C04662=1163.897,109.630,-53.464,-178.969,6.427,148.867
C04663=1163.902,109.381,-53.445,-178.972,6.425,148.867
C04664=1163.907,109.131,-53.426,-178.975,6.424,148.868
C04665=1163.912,108.882,-53.407,-178.977,6.423,148.868
C04666=1163.917,108.633,-53.389,-178.980,6.421,148.868
C04667=1163.921,108.384,-53.370,-178.982,6.419,148.869
C04668=1163.927,108.134,-53.352,-178.985,6.418,148.870
C04669=1163.931,107.885,-53.332,-178.988,6.417,148.870
C04670=1163.936,107.636,-53.314,-178.990,6.415,148.870
C04671=1163.941,107.387,-53.295,-178.993,6.414,148.871
C04672=1163.945,107.137,-53.277,-178.996,6.412,148.871
C04673=1163.951,106.888,-53.258,-178.998,6.411,148.872
C04674=1163.956,106.639,-53.240,-179.001,6.410,148.872
C04675=1163.961,106.370,-53.219,-179.004,6.408,148.873
C04676=1163.966,106.102,-53.199,-179.007,6.407,148.873
C04677=1163.971,105.834,-53.179,-179.010,6.405,148.874
C04678=1163.976,105.565,-53.160,-179.013,6.404,148.874
C04679=1163.981,105.316,-53.140,-179.016,6.402,148.875
C04680=1163.986,105.067,-53.122,-179.018,6.401,148.875
C04681=1163.991,104.818,-53.103,-179.021,6.400,148.876
C04682=1163.996,104.568,-53.084,-179.024,6.398,148.876
C04683=1164.001,104.319,-53.066,-179.026,6.396,148.877
C04684=1164.005,104.070,-53.048,-179.029,6.395,148.877
C04685=1164.010,103.821,-53.030,-179.032,6.394,148.878
C04686=1164.015,103.571,-53.011,-179.034,6.392,148.878
C04687=1164.020,103.322,-52.992,-179.037,6.391,148.878
C04688=1164.025,103.073,-52.974,-179.039,6.390,148.879
C04689=1164.030,102.823,-52.955,-179.043,6.388,148.879
C04690=1164.035,102.574,-52.937,-179.045,6.387,148.880
C04691=1164.039,102.325,-52.919,-179.047,6.386,148.880
C04692=1164.044,102.076,-52.901,-179.051,6.384,148.881
C04693=1164.049,101.826,-52.882,-179.053,6.383,148.881
C04694=1164.054,101.577,-52.864,-179.056,6.381,148.882
C04695=1164.059,101.328,-52.845,-179.058,6.380,148.882
C04696=1164.064,101.079,-52.827,-179.061,6.379,148.883
C04697=1164.068,100.829,-52.809,-179.064,6.377,148.883
C04698=1164.074,100.580,-52.790,-179.066,6.376,148.884
C04699=1164.079,100.330,-52.772,-179.069,6.375,148.884
C04700=1164.083,100.082,-52.753,-179.072,6.373,148.885
C04701=1164.088,99.833,-52.735,-179.074,6.372,148.885
C04702=1164.092,99.583,-52.717,-179.077,6.370,148.886
C04703=1164.098,99.333,-52.698,-179.080,6.369,148.886
C04704=1164.103,99.084,-52.680,-179.083,6.367,148.887
C04705=1164.108,98.835,-52.662,-179.085,6.366,148.887
C04706=1164.113,98.586,-52.644,-179.088,6.365,148.888
C04707=1164.117,98.337,-52.625,-179.091,6.363,148.888
C04708=1164.122,98.087,-52.607,-179.093,6.363,148.889
C04709=1164.127,97.838,-52.589,-179.096,6.361,148.889
C04710=1164.132,97.589,-52.571,-179.099,6.360,148.890
C04711=1164.137,97.340,-52.553,-179.101,6.359,148.890
C04712=1164.142,97.090,-52.535,-179.104,6.357,148.891
C04713=1164.146,96.840,-52.517,-179.107,6.356,148.891
C04714=1164.151,96.591,-52.499,-179.109,6.355,148.891
C04715=1164.156,96.342,-52.481,-179.112,6.353,148.892
C04716=1164.161,96.093,-52.463,-179.115,6.352,148.893
C04717=1164.166,95.844,-52.445,-179.117,6.351,148.893
C04718=1164.171,95.595,-52.427,-179.120,6.349,148.893
C04719=1164.175,95.345,-52.408,-179.123,6.348,148.894
C04720=1164.180,95.096,-52.390,-179.125,6.347,148.894
C04721=1164.185,94.846,-52.372,-179.128,6.345,148.895
C04722=1164.190,94.597,-52.354,-179.131,6.344,148.895
C04723=1164.195,94.348,-52.336,-179.134,6.343,148.896
C04724=1164.200,94.099,-52.318,-179.136,6.341,148.896
C04725=1164.205,93.850,-52.300,-179.139,6.340,148.897
C04726=1164.210,93.600,-52.282,-179.142,6.339,148.897
C04727=1164.214,93.350,-52.265,-179.144,6.337,148.898
C04728=1164.219,93.101,-52.247,-179.148,6.336,148.898
C04729=1164.224,92.852,-52.229,-179.150,6.335,148.899
C04730=1164.229,92.602,-52.211,-179.152,6.333,148.899
C04731=1164.234,92.353,-52.193,-179.156,6.332,148.900
C04732=1164.239,92.104,-52.175,-179.158,6.331,148.900
C04733=1164.244,91.855,-52.157,-179.160,6.329,148.901
C04734=1164.249,91.605,-52.140,-179.163,6.329,148.901
C04735=1164.254,91.356,-52.122,-179.166,6.327,148.902
C04736=1164.259,91.107,-52.104,-179.169,6.325,148.902
C04737=1164.264,90.858,-52.086,-179.171,6.325,148.903
C04738=1164.269,90.608,-52.068,-179.174,6.323,148.903
C04739=1164.274,90.359,-52.051,-179.177,6.322,148.904
C04740=1164.279,90.109,-52.033,-179.179,6.321,148.904
C04741=1164.284,89.860,-52.015,-179.182,6.319,148.905
C04742=1164.287,89.611,-51.997,-179.185,6.318,148.905
C04743=1164.292,89.361,-51.980,-179.187,6.317,148.906
C04744=1164.297,89.112,-51.962,-179.190,6.315,148.906
C04745=1164.302,88.863,-51.944,-179.192,6.315,148.907
C04746=1164.307,88.613,-51.926,-179.195,6.313,148.907
C04747=1164.312,88.364,-51.908,-179.198,6.311,148.908
C04748=1164.317,88.114,-51.890,-179.200,6.311,148.908
C04749=1164.322,87.865,-51.872,-179.203,6.309,148.909
C04750=1164.327,87.616,-51.856,-179.206,6.308,148.909
C04751=1164.332,87.367,-51.838,-179.208,6.307,148.910
C04752=1164.337,87.117,-51.820,-179.212,6.305,148.910
C04753=1164.342,86.868,-51.802,-179.214,6.304,148.911
C04754=1164.347,86.618,-51.785,-179.217,6.303,148.911
C04755=1164.352,86.369,-51.767,-179.220,6.301,148.912
C04756=1164.357,86.120,-51.750,-179.222,6.301,148.912
C04757=1164.362,85.871,-51.732,-179.225,6.299,148.913
C04758=1164.367,85.622,-51.715,-179.227,6.298,148.913
C04759=1164.372,85.372,-51.697,-179.230,6.297,148.914
C04760=1164.376,85.123,-51.680,-179.233,6.295,148.914
C04761=1164.381,84.874,-51.662,-179.235,6.294,148.915
C04762=1164.386,84.625,-51.644,-179.238,6.293,148.915
C04763=1164.391,84.375,-51.627,-179.241,6.292,148.916
C04764=1164.395,84.126,-51.610,-179.243,6.291,148.916
C04765=1164.401,83.876,-51.592,-179.246,6.290,148.917
C04766=1164.406,83.627,-51.574,-179.249,6.288,148.917
C04767=1164.411,83.377,-51.557,-179.251,6.287,148.918
C04768=1164.415,83.128,-51.540,-179.254,6.286,148.918
C04769=1164.420,82.878,-51.523,-179.257,6.284,148.919
C04770=1164.425,82.629,-51.505,-179.259,6.284,148.919
C04771=1164.430,82.380,-51.488,-179.262,6.282,148.920
C04772=1164.435,82.131,-51.470,-179.265,6.280,148.920
C04773=1164.440,81.881,-51.453,-179.267,6.280,148.921
C04774=1164.445,81.632,-51.436,-179.270,6.278,148.921
C04775=1164.450,81.383,-51.418,-179.272,6.277,148.922
C04776=1164.455,81.133,-51.401,-179.276,6.276,148.923
C04777=1164.459,80.884,-51.384,-179.278,6.275,148.923
C04778=1164.464,80.634,-51.366,-179.280,6.273,148.923
C04779=1164.470,80.366,-51.348,-179.284,6.272,148.924
C04780=1164.475,80.098,-51.329,-179.286,6.272,148.925
C04781=1164.480,79.829,-51.311,-179.289,6.270,148.925
C04782=1164.486,79.561,-51.292,-179.292,6.269,148.926
C04783=1164.490,79.312,-51.276,-179.295,6.267,148.926
C04784=1164.495,79.063,-51.258,-179.297,6.266,148.927
C04785=1164.501,78.813,-51.240,-179.300,6.265,148.927
C04786=1164.505,78.563,-51.224,-179.302,6.264,148.928
C04787=1164.510,78.314,-51.206,-179.306,6.263,148.928
C04788=1164.515,78.065,-51.189,-179.308,6.262,148.929
C04789=1164.520,77.816,-51.172,-179.311,6.260,148.929
C04790=1164.525,77.566,-51.155,-179.313,6.259,148.930
C04791=1164.530,77.317,-51.138,-179.316,6.258,148.930
C04792=1164.535,77.067,-51.120,-179.319,6.257,148.931
C04793=1164.540,76.818,-51.104,-179.321,6.256,148.931
C04794=1164.545,76.568,-51.087,-179.324,6.254,148.932
C04795=1164.549,76.320,-51.069,-179.327,6.253,148.932
C04796=1164.555,76.070,-51.052,-179.329,6.252,148.933
C04797=1164.559,75.820,-51.035,-179.332,6.251,148.934
C04798=1164.565,75.571,-51.018,-179.335,6.249,148.934
C04799=1164.569,75.322,-51.002,-179.337,6.249,148.934
C04800=1164.574,75.073,-50.984,-179.340,6.247,148.935
C04801=1164.579,74.823,-50.967,-179.342,6.246,148.935
C04802=1164.585,74.574,-50.950,-179.345,6.245,148.936
C04803=1164.589,74.325,-50.934,-179.348,6.244,148.937
C04804=1164.594,74.075,-50.916,-179.350,6.242,148.937
C04805=1164.599,73.825,-50.900,-179.353,6.242,148.938
C04806=1164.605,73.576,-50.883,-179.356,6.240,148.938
C04807=1164.609,73.327,-50.866,-179.358,6.240,148.939
C04808=1164.614,73.077,-50.848,-179.361,6.238,148.939
C04809=1164.618,72.828,-50.831,-179.364,6.238,148.940
C04810=1164.624,72.579,-50.815,-179.366,6.236,148.940
C04811=1164.629,72.329,-50.798,-179.369,6.235,148.941
C04812=1164.633,72.080,-50.781,-179.372,6.234,148.941
C04813=1164.638,71.830,-50.764,-179.374,6.233,148.942
C04814=1164.644,71.581,-50.748,-179.377,6.232,148.942
C04815=1164.648,71.332,-50.731,-179.379,6.231,148.943
C04816=1164.653,71.082,-50.714,-179.382,6.229,148.944
C04817=1164.658,70.833,-50.697,-179.385,6.228,148.944
C04818=1164.664,70.584,-50.680,-179.387,6.227,148.944
C04819=1164.668,70.334,-50.663,-179.390,6.226,148.945
C04820=1164.673,70.085,-50.647,-179.393,6.225,148.945
C04821=1164.678,69.835,-50.630,-179.395,6.224,148.946
C04822=1164.683,69.586,-50.613,-179.398,6.222,148.947
C04823=1164.688,69.337,-50.597,-179.400,6.221,148.947
C04824=1164.693,69.087,-50.580,-179.403,6.220,148.948
C04825=1164.698,68.838,-50.563,-179.406,6.219,148.948
C04826=1164.703,68.589,-50.547,-179.409,6.218,148.949
C04827=1164.708,68.339,-50.530,-179.411,6.217,148.949
C04828=1164.713,68.089,-50.513,-179.414,6.216,148.950
C04829=1164.718,67.840,-50.497,-179.416,6.215,148.950
C04830=1164.722,67.591,-50.481,-179.420,6.214,148.951
C04831=1164.727,67.341,-50.463,-179.422,6.213,148.951
C04832=1164.732,67.092,-50.447,-179.424,6.211,148.952
C04833=1164.737,66.843,-50.430,-179.427,6.211,148.952
C04834=1164.742,66.593,-50.413,-179.430,6.209,148.953
C04835=1164.748,66.344,-50.397,-179.432,6.208,148.954
C04836=1164.752,66.094,-50.381,-179.435,6.207,148.954
C04837=1164.757,65.845,-50.364,-179.438,6.206,148.955
C04838=1164.762,65.596,-50.347,-179.441,6.204,148.955
C04839=1164.767,65.346,-50.331,-179.443,6.204,148.956
C04840=1164.772,65.097,-50.315,-179.446,6.202,148.956
C04841=1164.777,64.847,-50.298,-179.448,6.201,148.957
C04842=1164.782,64.598,-50.282,-179.451,6.201,148.957
C04843=1164.787,64.349,-50.265,-179.453,6.199,148.958
C04844=1164.792,64.099,-50.249,-179.456,6.199,148.958
C04845=1164.797,63.850,-50.232,-179.459,6.197,148.959
C04846=1164.801,63.600,-50.216,-179.461,6.197,148.959
C04847=1164.806,63.352,-50.199,-179.464,6.195,148.960
C04848=1164.812,63.101,-50.183,-179.467,6.194,148.961
C04849=1164.817,62.852,-50.167,-179.470,6.193,148.961
C04850=1164.822,62.603,-50.150,-179.472,6.192,148.961
C04851=1164.826,62.353,-50.134,-179.474,6.191,148.962
C04852=1164.831,62.104,-50.118,-179.477,6.190,148.963
C04853=1164.836,61.854,-50.101,-179.480,6.189,148.963
C04854=1164.841,61.605,-50.085,-179.482,6.187,148.964
C04855=1164.846,61.355,-50.068,-179.485,6.187,148.964
C04856=1164.852,61.107,-50.052,-179.488,6.185,148.965
C04857=1164.856,60.856,-50.036,-179.490,6.185,148.965
C04858=1164.861,60.608,-50.020,-179.493,6.183,148.966
C04859=1164.866,60.358,-50.004,-179.496,6.183,148.966
C04860=1164.871,60.109,-49.987,-179.498,6.182,148.967
C04861=1164.876,59.859,-49.971,-179.501,6.180,148.967
C04862=1164.881,59.610,-49.955,-179.503,6.180,148.968
C04863=1164.886,59.360,-49.938,-179.506,6.178,148.968
C04864=1164.891,59.111,-49.923,-179.509,6.177,148.969
C04865=1164.895,58.861,-49.906,-179.512,6.176,148.970
C04866=1164.902,58.612,-49.890,-179.514,6.175,148.970
C04867=1164.906,58.362,-49.873,-179.516,6.174,148.971
C04868=1164.911,58.113,-49.858,-179.520,6.173,148.971
C04869=1164.916,57.863,-49.841,-179.522,6.172,148.972
C04870=1164.921,57.614,-49.825,-179.525,6.171,148.972
C04871=1164.926,57.364,-49.809,-179.527,6.170,148.973
C04872=1164.931,57.115,-49.793,-179.530,6.169,148.974
C04873=1164.936,56.866,-49.777,-179.532,6.168,148.974
C04874=1164.941,56.616,-49.761,-179.535,6.167,148.975
C04875=1164.946,56.367,-49.745,-179.538,6.166,148.975
C04876=1164.951,56.117,-49.729,-179.540,6.165,148.976
C04877=1164.956,55.869,-49.712,-179.543,6.164,148.976
C04878=1164.961,55.618,-49.696,-179.546,6.163,148.977
C04879=1164.966,55.370,-49.680,-179.548,6.162,148.977
C04880=1164.971,55.120,-49.664,-179.551,6.160,148.978
C04881=1164.976,54.870,-49.649,-179.553,6.160,148.978
C04882=1164.981,54.621,-49.632,-179.556,6.159,148.979
C04883=1164.986,54.352,-49.615,-179.559,6.158,148.979
C04884=1164.992,54.084,-49.598,-179.562,6.156,148.980
C04885=1164.997,53.815,-49.581,-179.564,6.156,148.981
C04886=1165.003,53.547,-49.564,-179.567,6.154,148.981
C04887=1165.007,53.297,-49.549,-179.570,6.154,148.982
C04888=1165.012,53.048,-49.532,-179.573,6.152,148.982
C04889=1165.017,52.799,-49.517,-179.575,6.152,148.983
C04890=1165.022,52.549,-49.501,-179.578,6.151,148.983
C04891=1165.027,52.300,-49.484,-179.581,6.149,148.984
C04892=1165.032,52.050,-49.468,-179.583,6.149,148.985
C04893=1165.037,51.800,-49.453,-179.586,6.148,148.985
C04894=1165.042,51.552,-49.437,-179.588,6.146,148.986
C04895=1165.047,51.301,-49.421,-179.591,6.146,148.986
C04896=1165.052,51.052,-49.406,-179.594,6.144,148.987
C04897=1165.057,50.803,-49.390,-179.596,6.143,148.987
C04898=1165.062,50.554,-49.373,-179.598,6.143,148.988
C04899=1165.067,50.304,-49.358,-179.601,6.141,148.988
C04900=1165.072,50.055,-49.342,-179.604,6.141,148.989
C04901=1165.077,49.805,-49.326,-179.606,6.140,148.989
C04902=1165.082,49.556,-49.311,-179.609,6.139,148.990
C04903=1165.087,49.307,-49.295,-179.611,6.138,148.991
C04904=1165.092,49.057,-49.279,-179.614,6.137,148.991
C04905=1165.097,48.807,-49.263,-179.617,6.136,148.992
C04906=1165.102,48.558,-49.248,-179.619,6.135,148.992
C04907=1165.107,48.308,-49.232,-179.622,6.134,148.993
C04908=1165.112,48.059,-49.217,-179.625,6.133,148.993
C04909=1165.117,47.810,-49.201,-179.627,6.132,148.994
C04910=1165.122,47.560,-49.185,-179.630,6.131,148.995
C04911=1165.127,47.311,-49.170,-179.632,6.130,148.995
C04912=1165.132,47.061,-49.154,-179.635,6.129,148.996
C04913=1165.137,46.812,-49.138,-179.638,6.128,148.996
C04914=1165.142,46.562,-49.122,-179.640,6.127,148.997
C04915=1165.147,46.313,-49.107,-179.642,6.126,148.997
C04916=1165.152,46.063,-49.092,-179.646,6.125,148.998
C04917=1165.157,45.813,-49.076,-179.648,6.125,148.999
C04918=1165.162,45.564,-49.061,-179.651,6.124,148.999
C04919=1165.167,45.315,-49.045,-179.654,6.122,149.000
C04920=1165.172,45.065,-49.030,-179.656,6.122,149.000
C04921=1165.177,44.815,-49.014,-179.659,6.121,149.001
C04922=1165.182,44.566,-48.999,-179.661,6.119,149.001
C04923=1165.187,44.317,-48.983,-179.664,6.119,149.002
C04924=1165.193,44.067,-48.968,-179.666,6.118,149.002
C04925=1165.197,43.817,-48.952,-179.669,6.117,149.003
C04926=1165.202,43.568,-48.937,-179.671,6.116,149.003
C04927=1165.207,43.319,-48.921,-179.674,6.115,149.004
C04928=1165.212,43.070,-48.906,-179.677,6.114,149.005
C04929=1165.217,42.820,-48.890,-179.680,6.113,149.005
C04930=1165.222,42.570,-48.875,-179.682,6.112,149.006
C04931=1165.227,42.321,-48.860,-179.684,6.112,149.006
C04932=1165.232,42.072,-48.844,-179.687,6.110,149.007
C04933=1165.237,41.822,-48.829,-179.690,6.110,149.008
C04934=1165.242,41.573,-48.813,-179.692,6.109,149.008
C04935=1165.247,41.323,-48.797,-179.695,6.108,149.009
C04936=1165.252,41.074,-48.782,-179.697,6.107,149.009
C04937=1165.257,40.824,-48.768,-179.700,6.106,149.010
C04938=1165.262,40.575,-48.753,-179.703,6.105,149.010
C04939=1165.267,40.325,-48.737,-179.705,6.104,149.011
C04940=1165.273,40.076,-48.721,-179.707,6.103,149.011
C04941=1165.277,39.826,-48.706,-179.711,6.102,149.012
C04942=1165.282,39.577,-48.690,-179.713,6.101,149.012
C04943=1165.287,39.327,-48.676,-179.715,6.101,149.013
C04944=1165.293,39.078,-48.661,-179.718,6.100,149.014
C04945=1165.297,38.829,-48.646,-179.721,6.099,149.014
C04946=1165.303,38.579,-48.630,-179.724,6.098,149.015
C04947=1165.307,38.330,-48.615,-179.726,6.097,149.015
C04948=1165.312,38.079,-48.600,-179.729,6.096,149.016
C04949=1165.317,37.830,-48.585,-179.731,6.095,149.016
C04950=1165.322,37.581,-48.569,-179.734,6.095,149.017
C04951=1165.328,37.331,-48.554,-179.736,6.094,149.018
C04952=1165.333,37.082,-48.539,-179.739,6.092,149.018
C04953=1165.338,36.832,-48.524,-179.741,6.092,149.019
C04954=1165.343,36.583,-48.509,-179.744,6.091,149.019
C04955=1165.347,36.334,-48.494,-179.747,6.089,149.020
C04956=1165.353,36.084,-48.479,-179.749,6.089,149.021
C04957=1165.357,35.834,-48.464,-179.751,6.088,149.021
C04958=1165.363,35.585,-48.448,-179.754,6.088,149.022
C04959=1165.368,35.335,-48.434,-179.757,6.086,149.022
C04960=1165.373,35.086,-48.418,-179.759,6.085,149.023
C04961=1165.378,34.837,-48.403,-179.762,6.085,149.023
C04962=1165.383,34.587,-48.388,-179.765,6.083,149.024
C04963=1165.388,34.338,-48.373,-179.768,6.083,149.025
C04964=1165.393,34.088,-48.358,-179.770,6.082,149.025
C04965=1165.398,33.838,-48.343,-179.772,6.081,149.026
C04966=1165.403,33.589,-48.328,-179.775,6.080,149.026
C04967=1165.409,33.339,-48.313,-179.778,6.079,149.027
C04968=1165.413,33.090,-48.298,-179.780,6.079,149.027
C04969=1165.419,32.841,-48.283,-179.783,6.078,149.028
C04970=1165.424,32.591,-48.269,-179.785,6.076,149.028
C04971=1165.428,32.342,-48.254,-179.788,6.076,149.029
C04972=1165.434,32.092,-48.239,-179.790,6.075,149.029
C04973=1165.438,31.842,-48.223,-179.793,6.075,149.030
C04974=1165.443,31.593,-48.209,-179.795,6.073,149.031
C04975=1165.448,31.343,-48.194,-179.798,6.072,149.031
C04976=1165.453,31.093,-48.179,-179.801,6.072,149.032
C04977=1165.458,30.844,-48.164,-179.803,6.071,149.032
C04978=1165.464,30.594,-48.149,-179.806,6.070,149.033
C04979=1165.468,30.345,-48.134,-179.808,6.069,149.034
C04980=1165.473,30.096,-48.120,-179.811,6.068,149.034
C04981=1165.479,29.846,-48.105,-179.813,6.068,149.035
C04982=1165.484,29.596,-48.090,-179.816,6.066,149.035
C04983=1165.488,29.347,-48.075,-179.819,6.066,149.036
C04984=1165.494,29.097,-48.060,-179.821,6.065,149.036
C04985=1165.499,28.848,-48.045,-179.823,6.064,149.037
C04986=1165.503,28.599,-48.031,-179.826,6.064,149.038
C04987=1165.510,28.330,-48.015,-179.829,6.062,149.038
C04988=1165.515,28.061,-47.999,-179.832,6.062,149.039
C04989=1165.520,27.793,-47.984,-179.835,6.060,149.039
C04990=1165.526,27.523,-47.967,-179.837,6.060,149.040
C04991=1165.531,27.274,-47.953,-179.840,6.059,149.041
C04992=1165.536,27.025,-47.938,-179.842,6.058,149.041
C04993=1165.541,26.775,-47.924,-179.845,6.057,149.042
C04994=1165.546,26.525,-47.909,-179.847,6.056,149.042
C04995=1165.551,26.276,-47.894,-179.850,6.056,149.043
C04996=1165.556,26.026,-47.880,-179.852,6.055,149.044
C04997=1165.561,25.776,-47.865,-179.856,6.054,149.044
C04998=1165.566,25.527,-47.850,-179.858,6.053,149.045
C04999=1165.571,25.277,-47.836,-179.860,6.052,149.045
C05000=1165.576,25.028,-47.821,-179.863,6.052,149.046
C05001=1165.581,24.779,-47.807,-179.865,6.051,149.046
C05002=1165.586,24.529,-47.792,-179.868,6.050,149.047
C05003=1165.591,24.280,-47.778,-179.871,6.049,149.048
C05004=1165.597,24.030,-47.763,-179.873,6.049,149.048
C05005=1165.602,23.781,-47.748,-179.875,6.048,149.049
C05006=1165.607,23.531,-47.734,-179.878,6.047,149.049
C05007=1165.612,23.281,-47.720,-179.881,6.046,149.050
C05008=1165.617,23.031,-47.705,-179.883,6.045,149.051
C05009=1165.621,22.782,-47.690,-179.886,6.045,149.051
C05010=1165.626,22.533,-47.676,-179.888,6.044,149.052
C05011=1165.632,22.283,-47.662,-179.891,6.043,149.052
C05012=1165.637,22.034,-47.647,-179.894,6.042,149.053
C05013=1165.642,21.785,-47.632,-179.896,6.041,149.053
C05014=1165.647,21.535,-47.618,-179.898,6.040,149.054
C05015=1165.652,21.285,-47.604,-179.901,6.040,149.055
C05016=1165.657,21.035,-47.590,-179.903,6.039,149.055
C05017=1165.662,20.786,-47.575,-179.907,6.038,149.056
C05018=1165.667,20.537,-47.561,-179.909,6.037,149.056
C05019=1165.672,20.287,-47.547,-179.911,6.036,149.057
C05020=1165.677,20.038,-47.532,-179.914,6.036,149.058
C05021=1165.682,19.788,-47.518,-179.916,6.035,149.058
C05022=1165.688,19.538,-47.503,-179.919,6.035,149.059
C05023=1165.693,19.288,-47.489,-179.922,6.033,149.059
C05024=1165.698,19.039,-47.475,-179.924,6.033,149.060
C05025=1165.703,18.790,-47.461,-179.927,6.032,149.061
C05026=1165.708,18.540,-47.446,-179.929,6.031,149.061
C05027=1165.713,18.290,-47.432,-179.932,6.031,149.062
C05028=1165.718,18.041,-47.418,-179.934,6.030,149.062
C05029=1165.724,17.792,-47.404,-179.937,6.029,149.063
C05030=1165.728,17.542,-47.390,-179.939,6.028,149.063
C05031=1165.733,17.292,-47.375,-179.942,6.027,149.064
C05032=1165.738,17.043,-47.360,-179.945,6.027,149.065
C05033=1165.743,16.793,-47.346,-179.947,6.026,149.065
C05034=1165.749,16.544,-47.332,-179.949,6.026,149.066
C05035=1165.754,16.295,-47.318,-179.952,6.024,149.066
C05036=1165.759,16.045,-47.303,-179.955,6.023,149.067
C05037=1165.764,15.795,-47.290,-179.957,6.023,149.067
C05038=1165.769,15.546,-47.276,-179.960,6.022,149.068
C05039=1165.774,15.296,-47.262,-179.962,6.022,149.069
C05040=1165.779,15.046,-47.247,-179.964,6.021,149.069
C05041=1165.783,14.797,-47.234,-179.967,6.020,149.070
C05042=1165.789,14.548,-47.220,-179.970,6.019,149.070
C05043=1165.794,14.298,-47.206,-179.972,6.018,149.071
C05044=1165.799,14.048,-47.191,-179.975,6.017,149.071
C05045=1165.804,13.799,-47.177,-179.977,6.017,149.072
C05046=1165.809,13.550,-47.163,-179.980,6.017,149.073
C05047=1165.814,13.300,-47.149,-179.982,6.016,149.073
C05048=1165.819,13.050,-47.135,-179.985,6.015,149.074
C05049=1165.825,12.801,-47.121,-179.987,6.014,149.074
C05050=1165.830,12.551,-47.107,-179.990,6.013,149.075
C05051=1165.835,12.301,-47.093,-179.992,6.012,149.076
C05052=1165.839,12.052,-47.079,-179.995,6.012,149.076
C05053=1165.845,11.803,-47.065,-179.998,6.011,149.077
C05054=1165.850,11.553,-47.051,-180.000,6.010,149.077
C05055=1165.855,11.303,-47.037,179.998,6.010,149.078
C05056=1165.860,11.054,-47.023,179.995,6.009,149.079
C05057=1165.866,10.804,-47.009,179.992,6.008,149.079
C05058=1165.871,10.554,-46.995,179.990,6.007,149.080
C05059=1165.875,10.306,-46.982,179.987,6.007,149.080
C05060=1165.880,10.056,-46.967,179.985,6.006,149.081
C05061=1165.886,9.806,-46.954,179.983,6.005,149.082
C05062=1165.891,9.557,-46.940,179.980,6.005,149.082
C05063=1165.896,9.307,-46.926,179.978,6.004,149.083
C05064=1165.901,9.057,-46.911,179.975,6.004,149.083
C05065=1165.906,8.808,-46.899,179.972,6.002,149.084
C05066=1165.911,8.558,-46.884,179.970,6.001,149.084
C05067=1165.916,8.308,-46.870,179.967,6.001,149.085
C05068=1165.922,8.059,-46.856,179.965,6.000,149.086
C05069=1165.926,7.809,-46.843,179.962,6.000,149.086
C05070=1165.931,7.560,-46.829,179.960,5.999,149.087
C05071=1165.937,7.311,-46.815,179.957,5.998,149.087
C05072=1165.942,7.060,-46.802,179.955,5.998,149.088
C05073=1165.947,6.812,-46.788,179.953,5.997,149.089
C05074=1165.952,6.562,-46.774,179.949,5.996,149.089
C05075=1165.957,6.312,-46.760,179.947,5.995,149.090
C05076=1165.963,6.063,-46.746,179.944,5.995,149.090
C05077=1165.967,5.813,-46.733,179.942,5.994,149.091
C05078=1165.972,5.563,-46.719,179.940,5.993,149.092
C05079=1165.978,5.314,-46.705,179.937,5.993,149.092
C05080=1165.983,5.064,-46.691,179.935,5.992,149.093
C05081=1165.988,4.815,-46.678,179.932,5.992,149.093
C05082=1165.993,4.565,-46.664,179.930,5.991,149.094
C05083=1165.998,4.315,-46.651,179.927,5.990,149.095
C05084=1166.003,4.066,-46.637,179.925,5.990,149.095
C05085=1166.008,3.816,-46.623,179.922,5.988,149.096
C05086=1166.014,3.567,-46.610,179.919,5.988,149.096
C05087=1166.018,3.317,-46.596,179.917,5.987,149.097
C05088=1166.024,3.068,-46.583,179.914,5.986,149.098
C05089=1166.029,2.818,-46.569,179.912,5.986,149.098
C05090=1166.034,2.569,-46.556,179.910,5.985,149.099
C05091=1166.039,2.299,-46.541,179.907,5.985,149.099
C05092=1166.045,2.030,-46.526,179.904,5.984,149.100
C05093=1166.050,1.760,-46.511,179.902,5.983,149.101
C05094=1166.056,1.491,-46.498,179.899,5.982,149.101
C05095=1166.061,1.242,-46.483,179.896,5.982,149.102
C05096=1166.066,0.992,-46.470,179.894,5.981,149.102
C05097=1166.071,0.743,-46.457,179.891,5.980,149.103
C05098=1166.076,0.493,-46.443,179.889,5.980,149.104
C05099=1166.081,0.243,-46.429,179.887,5.979,149.104
C05100=1166.086,-0.007,-46.416,179.884,5.979,149.105
C05101=1166.091,-0.256,-46.402,179.882,5.978,149.105
C05102=1166.096,-0.506,-46.389,179.879,5.977,149.106
C05103=1166.102,-0.755,-46.376,179.877,5.977,149.107
C05104=1166.106,-1.005,-46.362,179.874,5.976,149.107
C05105=1166.112,-1.254,-46.349,179.871,5.975,149.108
C05106=1166.118,-1.503,-46.335,179.869,5.974,149.108
C05107=1166.122,-1.753,-46.322,179.866,5.974,149.109
C05108=1166.128,-2.003,-46.309,179.864,5.973,149.110
C05109=1166.132,-2.252,-46.295,179.861,5.972,149.110
C05110=1166.138,-2.502,-46.282,179.859,5.972,149.111
C05111=1166.142,-2.752,-46.269,179.857,5.971,149.111
C05112=1166.148,-3.001,-46.255,179.854,5.971,149.112
C05113=1166.153,-3.251,-46.242,179.852,5.970,149.113
C05114=1166.158,-3.501,-46.229,179.849,5.969,149.113
C05115=1166.163,-3.750,-46.216,179.846,5.969,149.114
C05116=1166.169,-4.000,-46.202,179.844,5.968,149.114
C05117=1166.173,-4.250,-46.189,179.842,5.968,149.115
C05118=1166.179,-4.499,-46.175,179.839,5.967,149.116
C05119=1166.184,-4.748,-46.163,179.837,5.966,149.116
C05120=1166.189,-4.998,-46.149,179.835,5.965,149.117
C05121=1166.194,-5.248,-46.137,179.832,5.965,149.117
C05122=1166.199,-5.497,-46.122,179.829,5.965,149.118
C05123=1166.204,-5.747,-46.110,179.827,5.964,149.118
C05124=1166.209,-5.997,-46.097,179.824,5.963,149.119
C05125=1166.215,-6.246,-46.084,179.822,5.962,149.120
C05126=1166.219,-6.495,-46.070,179.820,5.962,149.120
C05127=1166.225,-6.745,-46.057,179.817,5.962,149.121
C05128=1166.230,-6.995,-46.044,179.815,5.961,149.122
C05129=1166.235,-7.245,-46.031,179.812,5.960,149.122
C05130=1166.240,-7.494,-46.017,179.810,5.959,149.123
C05131=1166.245,-7.743,-46.005,179.807,5.959,149.123
C05132=1166.250,-7.993,-45.991,179.805,5.959,149.124
C05133=1166.255,-8.243,-45.979,179.802,5.958,149.125
C05134=1166.261,-8.493,-45.965,179.799,5.956,149.125
C05135=1166.266,-8.742,-45.952,179.797,5.956,149.126
C05136=1166.271,-8.991,-45.939,179.794,5.955,149.126
C05137=1166.276,-9.241,-45.925,179.792,5.955,149.127
C05138=1166.281,-9.491,-45.913,179.790,5.954,149.128
C05139=1166.286,-9.740,-45.900,179.787,5.953,149.128
C05140=1166.291,-9.990,-45.887,179.785,5.953,149.129
C05141=1166.296,-10.240,-45.874,179.782,5.952,149.129
C05142=1166.301,-10.490,-45.861,179.780,5.951,149.130
C05143=1166.307,-10.739,-45.848,179.777,5.951,149.131
C05144=1166.312,-10.989,-45.835,179.775,5.950,149.131
C05145=1166.316,-11.239,-45.822,179.772,5.950,149.132
C05146=1166.322,-11.488,-45.808,179.770,5.949,149.132
C05147=1166.327,-11.737,-45.796,179.768,5.948,149.133
C05148=1166.332,-11.987,-45.783,179.765,5.948,149.134
C05149=1166.338,-12.237,-45.770,179.762,5.947,149.134
C05150=1166.343,-12.486,-45.757,179.760,5.947,149.135
C05151=1166.347,-12.736,-45.744,179.757,5.946,149.135
C05152=1166.352,-12.985,-45.732,179.755,5.945,149.136
C05153=1166.358,-13.235,-45.718,179.753,5.945,149.137
C05154=1166.363,-13.484,-45.706,179.750,5.945,149.137
C05155=1166.368,-13.734,-45.693,179.748,5.944,149.138
C05156=1166.374,-13.984,-45.680,179.746,5.944,149.138
C05157=1166.379,-14.233,-45.667,179.743,5.943,149.139
C05158=1166.383,-14.483,-45.654,179.741,5.943,149.140
C05159=1166.388,-14.733,-45.641,179.738,5.942,149.140
C05160=1166.394,-14.982,-45.628,179.736,5.942,149.141
C05161=1166.399,-15.232,-45.616,179.733,5.941,149.141
C05162=1166.404,-15.482,-45.603,179.731,5.940,149.142
C05163=1166.409,-15.731,-45.591,179.728,5.940,149.143
C05164=1166.415,-15.981,-45.578,179.726,5.939,149.143
C05165=1166.420,-16.230,-45.565,179.724,5.939,149.144
C05166=1166.425,-16.480,-45.552,179.721,5.938,149.144
C05167=1166.430,-16.730,-45.539,179.719,5.937,149.145
C05168=1166.435,-16.979,-45.527,179.716,5.937,149.146
C05169=1166.440,-17.228,-45.514,179.714,5.936,149.146
C05170=1166.446,-17.479,-45.501,179.711,5.936,149.147
C05171=1166.451,-17.729,-45.489,179.709,5.935,149.147
C05172=1166.456,-17.978,-45.476,179.706,5.934,149.148
C05173=1166.461,-18.227,-45.464,179.704,5.934,149.149
C05174=1166.466,-18.477,-45.451,179.702,5.933,149.149
C05175=1166.471,-18.727,-45.438,179.699,5.933,149.150
C05176=1166.477,-18.976,-45.425,179.696,5.932,149.150
C05177=1166.482,-19.226,-45.413,179.694,5.931,149.151
C05178=1166.487,-19.476,-45.400,179.691,5.931,149.152
C05179=1166.492,-19.726,-45.387,179.689,5.930,149.152
C05180=1166.497,-19.975,-45.375,179.687,5.930,149.153
C05181=1166.502,-20.224,-45.362,179.684,5.929,149.153
C05182=1166.507,-20.474,-45.350,179.682,5.928,149.154
C05183=1166.513,-20.724,-45.337,179.679,5.928,149.155
C05184=1166.518,-20.974,-45.324,179.678,5.928,149.155
C05185=1166.523,-21.223,-45.311,179.675,5.928,149.156
C05186=1166.528,-21.473,-45.300,179.673,5.927,149.156
C05187=1166.534,-21.722,-45.287,179.670,5.926,149.157
C05188=1166.539,-21.972,-45.274,179.667,5.926,149.158
C05189=1166.543,-22.222,-45.261,179.665,5.925,149.158
C05190=1166.549,-22.472,-45.250,179.663,5.925,149.159
C05191=1166.554,-22.721,-45.237,179.660,5.924,149.159
C05192=1166.559,-22.970,-45.224,179.658,5.923,149.160
C05193=1166.564,-23.220,-45.212,179.655,5.923,149.161
C05194=1166.569,-23.469,-45.200,179.653,5.922,149.161
C05195=1166.575,-23.740,-45.186,179.650,5.922,149.162
C05196=1166.580,-24.010,-45.173,179.648,5.921,149.163
C05197=1166.586,-24.279,-45.159,179.645,5.921,149.163
C05198=1166.592,-24.550,-45.146,179.643,5.920,149.164
C05199=1166.597,-24.799,-45.133,179.640,5.920,149.164
C05200=1166.602,-25.048,-45.121,179.637,5.919,149.165
C05201=1166.608,-25.298,-45.109,179.635,5.918,149.166
C05202=1166.613,-25.547,-45.096,179.633,5.918,149.166
C05203=1166.618,-25.797,-45.084,179.630,5.917,149.167
C05204=1166.623,-26.047,-45.071,179.628,5.917,149.167
C05205=1166.628,-26.297,-45.059,179.626,5.916,149.168
C05206=1166.633,-26.547,-45.047,179.623,5.915,149.169
C05207=1166.639,-26.796,-45.034,179.620,5.915,149.169
C05208=1166.643,-27.046,-45.023,179.619,5.915,149.170
C05209=1166.648,-27.295,-45.010,179.616,5.914,149.170
C05210=1166.654,-27.545,-44.998,179.614,5.914,149.171
C05211=1166.659,-27.794,-44.986,179.611,5.913,149.172
C05212=1166.664,-28.044,-44.974,179.608,5.913,149.172
C05213=1166.669,-28.293,-44.961,179.606,5.912,149.173
C05214=1166.674,-28.543,-44.948,179.604,5.912,149.174
C05215=1166.679,-28.793,-44.936,179.601,5.911,149.174
C05216=1166.685,-29.043,-44.924,179.599,5.910,149.175
C05217=1166.690,-29.293,-44.912,179.596,5.910,149.175
C05218=1166.695,-29.542,-44.899,179.595,5.910,149.176
C05219=1166.701,-29.792,-44.887,179.592,5.909,149.177
C05220=1166.706,-30.042,-44.876,179.590,5.909,149.177
C05221=1166.710,-30.291,-44.864,179.587,5.908,149.178
C05222=1166.716,-30.541,-44.852,179.585,5.907,149.178
C05223=1166.721,-30.790,-44.839,179.582,5.907,149.179
C05224=1166.726,-31.040,-44.827,179.580,5.907,149.180
C05225=1166.731,-31.289,-44.815,179.577,5.906,149.180
C05226=1166.737,-31.539,-44.803,179.575,5.905,149.181
C05227=1166.742,-31.789,-44.790,179.572,5.904,149.181
C05228=1166.747,-32.039,-44.778,179.570,5.905,149.182
C05229=1166.752,-32.288,-44.767,179.568,5.904,149.183
C05230=1166.757,-32.537,-44.754,179.566,5.904,149.183
C05231=1166.763,-32.787,-44.742,179.563,5.903,149.184
C05232=1166.768,-33.037,-44.731,179.561,5.902,149.184
C05233=1166.773,-33.287,-44.718,179.558,5.902,149.185
C05234=1166.779,-33.537,-44.706,179.556,5.901,149.185
C05235=1166.783,-33.786,-44.694,179.553,5.901,149.186
C05236=1166.788,-34.036,-44.682,179.551,5.900,149.187
C05237=1166.794,-34.286,-44.670,179.549,5.900,149.187
C05238=1166.799,-34.535,-44.658,179.546,5.900,149.188
C05239=1166.804,-34.785,-44.646,179.544,5.899,149.188
C05240=1166.809,-35.034,-44.635,179.541,5.899,149.189
C05241=1166.814,-35.284,-44.622,179.539,5.898,149.190
C05242=1166.820,-35.534,-44.610,179.537,5.897,149.190
C05243=1166.825,-35.784,-44.598,179.534,5.897,149.191
C05244=1166.830,-36.033,-44.587,179.532,5.897,149.192
C05245=1166.835,-36.283,-44.574,179.530,5.897,149.192
C05246=1166.840,-36.532,-44.562,179.528,5.896,149.193
C05247=1166.846,-36.782,-44.550,179.525,5.895,149.193
C05248=1166.850,-37.032,-44.539,179.522,5.895,149.194
C05249=1166.856,-37.281,-44.527,179.520,5.894,149.195
C05250=1166.861,-37.531,-44.515,179.517,5.894,149.195
C05251=1166.866,-37.781,-44.503,179.515,5.893,149.196
C05252=1166.872,-38.030,-44.492,179.513,5.893,149.196
C05253=1166.877,-38.279,-44.479,179.511,5.892,149.197
C05254=1166.882,-38.529,-44.467,179.508,5.892,149.198
C05255=1166.888,-38.779,-44.456,179.506,5.892,149.198
C05256=1166.892,-39.029,-44.444,179.503,5.891,149.199
C05257=1166.898,-39.279,-44.432,179.501,5.890,149.200
C05258=1166.903,-39.529,-44.420,179.499,5.889,149.200
C05259=1166.908,-39.778,-44.408,179.496,5.890,149.201
C05260=1166.913,-40.028,-44.397,179.494,5.889,149.201
C05261=1166.919,-40.278,-44.385,179.492,5.889,149.202
C05262=1166.923,-40.527,-44.373,179.489,5.888,149.203
C05263=1166.929,-40.777,-44.362,179.487,5.887,149.203
C05264=1166.935,-41.027,-44.350,179.484,5.887,149.204
C05265=1166.939,-41.275,-44.338,179.483,5.887,149.204
C05266=1166.945,-41.525,-44.326,179.480,5.887,149.205
C05267=1166.950,-41.775,-44.314,179.477,5.886,149.206
C05268=1166.955,-42.025,-44.303,179.475,5.885,149.206
C05269=1166.960,-42.275,-44.291,179.472,5.885,149.207
C05270=1166.965,-42.525,-44.280,179.470,5.884,149.207
C05271=1166.971,-42.774,-44.268,179.468,5.884,149.208
C05272=1166.976,-43.024,-44.256,179.466,5.884,149.208
C05273=1166.981,-43.273,-44.245,179.463,5.883,149.209
C05274=1166.986,-43.523,-44.233,179.461,5.883,149.210
C05275=1166.992,-43.773,-44.221,179.458,5.882,149.210
C05276=1166.996,-44.023,-44.210,179.456,5.882,149.211
C05277=1167.002,-44.273,-44.198,179.454,5.882,149.211
C05278=1167.007,-44.522,-44.187,179.451,5.881,149.212
C05279=1167.013,-44.772,-44.175,179.449,5.880,149.213
C05280=1167.017,-45.021,-44.164,179.447,5.880,149.213
C05281=1167.023,-45.271,-44.152,179.444,5.879,149.214
C05282=1167.028,-45.521,-44.140,179.442,5.879,149.215
C05283=1167.033,-45.771,-44.129,179.440,5.879,149.215
C05284=1167.039,-46.020,-44.117,179.438,5.878,149.216
C05285=1167.044,-46.270,-44.106,179.435,5.878,149.216
C05286=1167.049,-46.520,-44.094,179.433,5.877,149.217
C05287=1167.054,-46.769,-44.083,179.430,5.877,149.218
C05288=1167.059,-47.019,-44.071,179.428,5.877,149.218
C05289=1167.064,-47.268,-44.060,179.426,5.876,149.219
C05290=1167.070,-47.518,-44.048,179.423,5.876,149.219
C05291=1167.075,-47.768,-44.037,179.421,5.875,149.220
C05292=1167.080,-48.018,-44.025,179.418,5.875,149.221
C05293=1167.085,-48.266,-44.014,179.417,5.875,149.221
C05294=1167.091,-48.516,-44.002,179.414,5.874,149.222
C05295=1167.095,-48.766,-43.991,179.412,5.873,149.222
C05296=1167.101,-49.016,-43.979,179.409,5.873,149.223
C05297=1167.106,-49.266,-43.969,179.406,5.873,149.224
C05298=1167.112,-49.515,-43.957,179.404,5.872,149.224
C05299=1167.117,-49.786,-43.944,179.402,5.872,149.225
C05300=1167.123,-50.057,-43.932,179.400,5.872,149.226
C05301=1167.128,-50.327,-43.921,179.397,5.871,149.226
C05302=1167.134,-50.597,-43.908,179.395,5.871,149.227
C05303=1167.139,-50.847,-43.896,179.392,5.870,149.227
C05304=1167.145,-51.097,-43.885,179.390,5.869,149.228
C05305=1167.150,-51.347,-43.874,179.387,5.869,149.229
C05306=1167.155,-51.596,-43.862,179.386,5.869,149.229
C05307=1167.160,-51.846,-43.850,179.383,5.868,149.230
C05308=1167.165,-52.095,-43.839,179.380,5.868,149.231
C05309=1167.170,-52.345,-43.829,179.378,5.867,149.231
C05310=1167.176,-52.595,-43.817,179.375,5.867,149.232
C05311=1167.181,-52.844,-43.806,179.374,5.867,149.232
C05312=1167.187,-53.094,-43.794,179.371,5.866,149.233
C05313=1167.192,-53.344,-43.784,179.369,5.866,149.233
C05314=1167.196,-53.594,-43.772,179.366,5.865,149.234
C05315=1167.202,-53.843,-43.761,179.364,5.864,149.235
C05316=1167.207,-54.093,-43.750,179.362,5.865,149.235
C05317=1167.212,-54.343,-43.739,179.359,5.864,149.236
C05318=1167.218,-54.592,-43.727,179.357,5.864,149.236
C05319=1167.223,-54.842,-43.716,179.354,5.863,149.237
C05320=1167.227,-55.092,-43.705,179.353,5.863,149.238
C05321=1167.234,-55.341,-43.694,179.350,5.863,149.238
C05322=1167.238,-55.591,-43.683,179.348,5.862,149.239
C05323=1167.243,-55.841,-43.671,179.345,5.862,149.240
C05324=1167.249,-56.090,-43.661,179.343,5.861,149.240
C05325=1167.254,-56.340,-43.649,179.341,5.861,149.241
C05326=1167.259,-56.590,-43.638,179.339,5.860,149.241
C05327=1167.265,-56.840,-43.627,179.336,5.860,149.242
C05328=1167.270,-57.089,-43.616,179.334,5.860,149.243
C05329=1167.275,-57.339,-43.605,179.332,5.860,149.243
C05330=1167.281,-57.589,-43.594,179.329,5.859,149.244
C05331=1167.286,-57.838,-43.583,179.327,5.858,149.244
C05332=1167.290,-58.088,-43.571,179.324,5.858,149.245
C05333=1167.296,-58.337,-43.561,179.323,5.858,149.245
C05334=1167.301,-58.587,-43.549,179.320,5.858,149.246
C05335=1167.306,-58.838,-43.539,179.318,5.857,149.247
C05336=1167.312,-59.087,-43.528,179.315,5.856,149.247
C05337=1167.316,-59.336,-43.516,179.314,5.856,149.248
C05338=1167.322,-59.587,-43.505,179.311,5.856,149.248
C05339=1167.327,-59.836,-43.494,179.308,5.856,149.249
C05340=1167.332,-60.086,-43.484,179.306,5.855,149.250
C05341=1167.338,-60.335,-43.473,179.304,5.855,149.250
C05342=1167.343,-60.585,-43.462,179.302,5.854,149.251
C05343=1167.348,-60.835,-43.450,179.299,5.854,149.252
C05344=1167.354,-61.085,-43.440,179.297,5.853,149.252
C05345=1167.358,-61.334,-43.429,179.295,5.853,149.253
C05346=1167.365,-61.584,-43.418,179.293,5.853,149.253
C05347=1167.369,-61.834,-43.407,179.290,5.852,149.254
C05348=1167.374,-62.084,-43.396,179.288,5.851,149.254
C05349=1167.380,-62.333,-43.385,179.286,5.852,149.255
C05350=1167.385,-62.583,-43.375,179.284,5.851,149.256
C05351=1167.390,-62.832,-43.364,179.281,5.851,149.256
C05352=1167.396,-63.083,-43.353,179.278,5.850,149.257
C05353=1167.401,-63.332,-43.342,179.277,5.850,149.257
C05354=1167.406,-63.582,-43.331,179.274,5.850,149.258
C05355=1167.411,-63.831,-43.320,179.272,5.849,149.259
C05356=1167.416,-64.081,-43.310,179.269,5.849,149.259
C05357=1167.421,-64.331,-43.298,179.268,5.849,149.260
C05358=1167.427,-64.580,-43.288,179.265,5.848,149.261
C05359=1167.432,-64.831,-43.277,179.263,5.847,149.261
C05360=1167.438,-65.080,-43.266,179.261,5.848,149.262
C05361=1167.443,-65.330,-43.255,179.259,5.847,149.262
C05362=1167.448,-65.579,-43.245,179.256,5.847,149.263
C05363=1167.453,-65.829,-43.234,179.254,5.846,149.263
C05364=1167.458,-66.079,-43.223,179.252,5.846,149.264
C05365=1167.464,-66.328,-43.212,179.249,5.845,149.265
C05366=1167.469,-66.579,-43.201,179.247,5.845,149.265
C05367=1167.474,-66.828,-43.190,179.245,5.844,149.266
C05368=1167.479,-67.078,-43.180,179.243,5.845,149.266
C05369=1167.485,-67.327,-43.170,179.240,5.844,149.267
C05370=1167.489,-67.577,-43.158,179.238,5.844,149.268
C05371=1167.495,-67.827,-43.148,179.236,5.844,149.268
C05372=1167.500,-68.077,-43.138,179.233,5.843,149.269
C05373=1167.505,-68.326,-43.127,179.231,5.843,149.270
C05374=1167.510,-68.576,-43.116,179.229,5.842,149.270
C05375=1167.516,-68.826,-43.106,179.226,5.842,149.271
C05376=1167.521,-69.076,-43.094,179.224,5.842,149.271
C05377=1167.527,-69.325,-43.084,179.222,5.841,149.272
C05378=1167.532,-69.575,-43.073,179.220,5.841,149.272
C05379=1167.538,-69.825,-43.063,179.217,5.841,149.273
C05380=1167.543,-70.074,-43.052,179.215,5.840,149.274
C05381=1167.548,-70.324,-43.041,179.212,5.840,149.274
C05382=1167.553,-70.574,-43.031,179.211,5.840,149.275
C05383=1167.558,-70.824,-43.021,179.208,5.839,149.276
C05384=1167.564,-71.073,-43.010,179.206,5.838,149.276
C05385=1167.569,-71.323,-42.999,179.204,5.839,149.277
C05386=1167.574,-71.573,-42.989,179.202,5.838,149.277
C05387=1167.579,-71.823,-42.978,179.199,5.838,149.278
C05388=1167.585,-72.072,-42.967,179.198,5.838,149.278
C05389=1167.590,-72.322,-42.957,179.195,5.837,149.279
C05390=1167.595,-72.571,-42.947,179.193,5.836,149.280
C05391=1167.601,-72.821,-42.936,179.190,5.836,149.280
C05392=1167.606,-73.071,-42.926,179.188,5.836,149.281
C05393=1167.611,-73.320,-42.915,179.186,5.836,149.281
C05394=1167.616,-73.570,-42.904,179.184,5.835,149.282
C05395=1167.622,-73.820,-42.894,179.181,5.835,149.283
C05396=1167.627,-74.070,-42.884,179.179,5.834,149.283
C05397=1167.632,-74.320,-42.873,179.177,5.834,149.284
C05398=1167.638,-74.569,-42.863,179.175,5.834,149.284
C05399=1167.643,-74.820,-42.853,179.172,5.834,149.285
C05400=1167.648,-75.068,-42.842,179.170,5.833,149.285
C05401=1167.654,-75.318,-42.831,179.168,5.833,149.286
C05402=1167.658,-75.568,-42.821,179.166,5.832,149.287
C05403=1167.664,-75.840,-42.810,179.163,5.832,149.287
C05404=1167.671,-76.110,-42.799,179.161,5.832,149.288
C05405=1167.676,-76.382,-42.788,179.158,5.831,149.289
C05406=1167.682,-76.653,-42.776,179.156,5.831,149.289
C05407=1167.687,-76.903,-42.766,179.154,5.831,149.290
C05408=1167.692,-77.151,-42.756,179.151,5.830,149.290
C05409=1167.697,-77.402,-42.745,179.149,5.831,149.291
C05410=1167.702,-77.651,-42.735,179.147,5.830,149.292
C05411=1167.708,-77.901,-42.725,179.144,5.829,149.292
C05412=1167.713,-78.151,-42.714,179.143,5.829,149.293
C05413=1167.719,-78.401,-42.704,179.140,5.829,149.294
C05414=1167.724,-78.650,-42.694,179.138,5.828,149.294
C05415=1167.729,-78.900,-42.683,179.136,5.829,149.295
C05416=1167.735,-79.150,-42.673,179.134,5.828,149.295
C05417=1167.740,-79.399,-42.663,179.131,5.827,149.296
C05418=1167.745,-79.649,-42.653,179.129,5.827,149.296
C05419=1167.750,-79.899,-42.643,179.127,5.827,149.297
C05420=1167.756,-80.149,-42.632,179.125,5.826,149.298
C05421=1167.761,-80.399,-42.622,179.123,5.827,149.298
C05422=1167.766,-80.648,-42.612,179.120,5.826,149.299
C05423=1167.771,-80.898,-42.602,179.118,5.825,149.300
C05424=1167.776,-81.148,-42.591,179.116,5.825,149.300
C05425=1167.782,-81.397,-42.581,179.114,5.825,149.300
C05426=1167.787,-81.647,-42.571,179.111,5.824,149.301
C05427=1167.792,-81.897,-42.560,179.110,5.824,149.302
C05428=1167.798,-82.147,-42.552,179.107,5.824,149.302
C05429=1167.803,-82.397,-42.541,179.105,5.823,149.303
C05430=1167.808,-82.647,-42.531,179.103,5.824,149.304
C05431=1167.814,-82.896,-42.521,179.100,5.823,149.304
C05432=1167.819,-83.146,-42.510,179.098,5.822,149.305
C05433=1167.824,-83.396,-42.500,179.096,5.822,149.305
C05434=1167.829,-83.645,-42.490,179.094,5.822,149.306
C05435=1167.835,-83.895,-42.480,179.091,5.821,149.306
C05436=1167.840,-84.144,-42.470,179.089,5.822,149.307
C05437=1167.845,-84.394,-42.460,179.087,5.821,149.308
C05438=1167.851,-84.645,-42.450,179.084,5.820,149.308
C05439=1167.856,-84.894,-42.440,179.083,5.820,149.309
C05440=1167.861,-85.143,-42.430,179.080,5.820,149.310
C05441=1167.866,-85.394,-42.420,179.079,5.820,149.310
C05442=1167.872,-85.643,-42.410,179.076,5.820,149.311
C05443=1167.877,-85.893,-42.399,179.074,5.819,149.311
C05444=1167.882,-86.143,-42.390,179.072,5.819,149.312
C05445=1167.887,-86.393,-42.380,179.069,5.818,149.312
C05446=1167.893,-86.642,-42.370,179.067,5.818,149.313
C05447=1167.898,-86.891,-42.360,179.065,5.818,149.314
C05448=1167.903,-87.142,-42.350,179.063,5.817,149.314
C05449=1167.909,-87.392,-42.340,179.060,5.817,149.315
C05450=1167.914,-87.641,-42.330,179.059,5.817,149.315
C05451=1167.919,-87.891,-42.320,179.056,5.817,149.316
C05452=1167.925,-88.140,-42.310,179.054,5.817,149.316
C05453=1167.930,-88.390,-42.299,179.052,5.816,149.317
C05454=1167.935,-88.640,-42.291,179.050,5.815,149.318
C05455=1167.941,-88.890,-42.280,179.047,5.816,149.318
C05456=1167.945,-89.139,-42.271,179.045,5.815,149.319
C05457=1167.950,-89.389,-42.260,179.043,5.814,149.319
C05458=1167.956,-89.639,-42.251,179.041,5.815,149.320
C05459=1167.961,-89.889,-42.241,179.039,5.814,149.321
C05460=1167.967,-90.138,-42.231,179.037,5.814,149.321
C05461=1167.973,-90.388,-42.221,179.035,5.814,149.322
C05462=1167.977,-90.638,-42.211,179.032,5.813,149.322
C05463=1167.983,-90.888,-42.201,179.030,5.813,149.323
C05464=1167.989,-91.138,-42.192,179.028,5.813,149.324
C05465=1167.993,-91.387,-42.182,179.025,5.812,149.324
C05466=1167.999,-91.637,-42.172,179.024,5.812,149.325
C05467=1168.004,-91.887,-42.163,179.021,5.812,149.325
C05468=1168.009,-92.137,-42.152,179.020,5.812,149.326
C05469=1168.015,-92.386,-42.142,179.017,5.811,149.327
C05470=1168.020,-92.636,-42.133,179.015,5.810,149.327
C05471=1168.026,-92.886,-42.123,179.013,5.811,149.328
C05472=1168.030,-93.135,-42.113,179.010,5.810,149.328
C05473=1168.036,-93.385,-42.104,179.008,5.811,149.329
C05474=1168.041,-93.635,-42.094,179.006,5.810,149.329
C05475=1168.046,-93.885,-42.084,179.004,5.809,149.330
C05476=1168.052,-94.135,-42.074,179.002,5.809,149.331
C05477=1168.057,-94.384,-42.065,179.000,5.809,149.331
C05478=1168.063,-94.634,-42.055,178.998,5.809,149.332
C05479=1168.068,-94.884,-42.046,178.995,5.808,149.332
C05480=1168.074,-95.134,-42.036,178.993,5.808,149.333
C05481=1168.078,-95.384,-42.026,178.991,5.808,149.333
C05482=1168.083,-95.633,-42.016,178.989,5.807,149.334
C05483=1168.089,-95.883,-42.007,178.987,5.808,149.335
C05484=1168.094,-96.133,-41.997,178.985,5.807,149.335
C05485=1168.099,-96.382,-41.988,178.982,5.806,149.336
C05486=1168.105,-96.632,-41.978,178.980,5.806,149.336
C05487=1168.110,-96.882,-41.969,178.978,5.806,149.337
C05488=1168.116,-97.131,-41.959,178.976,5.806,149.338
C05489=1168.120,-97.382,-41.949,178.974,5.805,149.338
C05490=1168.126,-97.631,-41.939,178.971,5.805,149.339
C05491=1168.131,-97.881,-41.930,178.970,5.805,149.339
C05492=1168.137,-98.131,-41.920,178.967,5.804,149.340
C05493=1168.142,-98.381,-41.911,178.965,5.805,149.340
C05494=1168.147,-98.630,-41.901,178.963,5.804,149.341
C05495=1168.153,-98.880,-41.892,178.961,5.803,149.342
